Yaskawa INFORM job: OK_R2_O57-69(2)(90,0)_OK.JBI

/JOB
//NAME OK_R2_O57-69(2)(90,0)_OK
///FOLDERNAME X4
//POS
///NPOS 521,521,521,19,0,0
///TOOL 0
///POSTYPE PULSE
///PULSE
C00000=-135424,72899,29147,-3537,85342,3792
C00001=-134013,95021,61136,-4029,77105,4505
C00002=-134047,101087,71818,-4077,73656,4607
C00003=-134047,101216,72822,-4088,73105,4626
C00004=-134047,101094,71866,-4078,73630,4609
C00005=-133936,105187,77198,-4137,72460,4688
C00006=-134047,101094,71866,-4078,73630,4609
C00007=-133891,92563,58880,-4064,77236,4542
C00008=-133627,85963,47659,-4101,80754,4516
C00009=-133192,78294,50454,-10127,76922,11696
C00010=-133849,85255,61933,-10093,73405,11757
C00011=-135353,87618,67605,-9788,70974,11422
C00012=-135353,87997,69106,-9827,70255,11481
C00013=-135353,87618,67605,-9788,70974,11422
C00014=-135153,93739,75342,-9940,69404,11624
C00015=-135353,87618,67605,-9788,70974,11422
C00016=-133639,83161,60388,-10158,73308,11840
C00017=-132974,76301,49087,-10194,76769,11784
C00018=-129415,62996,33414,-11066,79991,12732
C00019=-98130,32671,61537,-45409,44339,32891
C00020=-100023,41688,73231,-46965,41628,33506
C00021=-100756,49088,84228,-49401,39255,34803
C00022=-100756,52120,89278,-50881,38240,35655
C00023=-100756,49088,84228,-49401,39255,34803
C00024=-101219,51120,86580,-49709,38764,34882
C00025=-100756,49088,84228,-49401,39255,34803
C00026=-97195,31965,62320,-46227,44186,33575
C00027=-75566,-2034,22500,-42402,86688,50389
C00028=-92276,-18388,7402,-33699,73725,46550
C00029=-92276,-17400,9548,-33822,73042,46763
C00030=-92276,-17933,8393,-33755,73407,46648
C00031=-120131,-32698,-12117,4829,66200,34356
C00032=-120131,-32114,-10702,4851,65630,34332
C00033=-120989,-32117,-10704,5006,65680,34020
C00034=-120131,-32114,-10702,4851,65630,34332
C00035=-120131,-38085,-26806,4645,72450,34604
C00036=-99101,-76935,-92016,-31014,74911,20401
C00037=-52587,-144740,-101483,-60524,64363,-65274
C00038=-46989,-65360,-59229,-62781,73103,-77672
C00039=-56832,-65466,-56421,-59287,64983,-77772
C00040=-57148,-65688,-55453,-59188,64110,-77279
C00041=-55649,-62097,-53047,-61106,66880,-78547
C00042=-57237,-59710,-51792,-60669,66110,-79037
C00043=-56277,-61326,-53166,-60831,66721,-78866
C00044=-55441,-62561,-53810,-61057,67127,-78609
C00045=-56207,-63985,-54541,-61032,66503,-78630
C00046=-55438,-62578,-53813,-61060,67126,-78606
C00047=-51973,-62323,-54701,-62406,69323,-78001
C00048=-48054,-62529,-57040,-62601,72472,-77896
C00049=-29811,-70761,-60283,-66780,94863,-53671
C00050=-30965,-22538,-31531,-67696,97011,-56857
C00051=-55044,-42598,-44870,-68563,88788,-43678
C00052=-56249,-45120,-46406,-68472,87844,-43687
C00053=-57925,-45354,-44812,-68371,86292,-43442
C00054=-57925,-45174,-43802,-68390,86084,-43215
C00055=-57925,-45354,-44812,-68371,86292,-43442
C00056=-59167,-45210,-44726,-68282,85469,-43617
C00057=-57925,-45354,-44812,-68371,86292,-43442
C00058=-55819,-44223,-45863,-68504,88181,-43684
C00059=-44722,-31045,-43816,-69927,97696,-44632
C00060=-43071,-26445,-40665,-70170,98951,-44614
C00061=-127706,-49493,-81773,19458,97242,-49666
C00062=-127020,6423,-39070,7004,99714,-51816
C00063=-127020,5137,-37554,6966,98131,-51906
C00064=-128416,4382,-35850,7239,96821,-52416
C00065=-128416,3847,-35017,7224,96041,-52460
C00066=-128416,4148,-35496,7233,96488,-52435
C00067=-130041,4566,-35136,7580,96617,-52937
C00068=-129924,4205,-34639,7545,96120,-52933
C00069=-129457,4078,-34747,7447,96082,-52788
C00070=-130190,4712,-35256,7614,96778,-52976
C00071=-128966,36168,-17458,7491,101844,-52285
C00072=-149392,-6912,-25974,9982,75562,-31317
C00073=-149173,-488,-12666,10148,70714,-31647
C00074=-149173,-326,-10897,10208,69722,-31733
C00075=-149173,-394,-11578,10184,70101,-31701
C00076=-148123,2416,-9216,9823,69962,-31333
C00077=-149173,-394,-11578,10184,70101,-31701
C00078=-152478,4885,-6741,15795,72623,-37698
C00079=-151455,3828,-7649,15488,72442,-37350
C00080=-152478,4560,-12614,15554,75946,-37261
C00081=-146445,-24647,-43161,13522,78564,-34847
C00082=-131494,-80468,-98534,7816,92108,-53678
C00083=-52065,-14099,-27709,-42253,108676,27596
C00084=-76671,-130461,-121705,-35735,90710,50834
C00085=-94829,-93442,-100428,-28991,96183,47377
C00086=-110716,-92055,-82664,-19311,98038,51285
C00087=-114275,-93352,-80055,-19461,95045,50478
C00088=-118122,-92212,-76367,-19656,92534,49497
C00089=-118129,-91398,-74848,-19645,92046,49575
C00090=-118122,-92212,-76367,-19656,92534,49497
C00091=-119808,-92271,-76389,-19753,92113,48959
C00092=-118122,-92212,-76367,-19656,92534,49497
C00093=-114499,-91094,-78376,-19482,95112,50387
C00094=-110992,-89821,-80983,-19339,98080,51178
C00095=-124454,-89651,-86550,11137,94998,-69701
C00096=-122569,-92184,-83910,11067,91866,-69331
C00097=-120652,-93960,-80852,11027,88857,-68936
C00098=-120652,-93520,-79457,11027,88237,-68992
C00099=-120652,-93960,-80852,11027,88857,-68936
C00100=-120650,-97396,-81866,11026,87737,-69033
C00101=-120652,-93960,-80852,11027,88857,-68936
C00102=-118161,-93768,-80427,10994,88357,-68121
C00103=-120652,-93960,-80852,11027,88857,-68936
C00104=-120037,-91891,-82714,11032,90945,-68539
C00105=-121981,-89592,-85452,11099,94026,-68936
C00106=-122005,-89480,-97857,11363,101580,-68254
C00107=-122005,-89427,-98101,11372,101754,-68238
C00108=-119094,-95812,-115555,-4544,90851,-20867
C00109=-116502,-111480,-109655,-18779,62868,21987
C00110=-119472,-101923,-104261,-17094,63743,20698
C00111=-121534,-96097,-100090,-16016,63743,19914
C00112=-121534,-96194,-98882,-16123,62979,20025
C00113=-112336,-84014,-94514,-26506,72534,27449
C00114=-114298,-84401,-94682,-25743,71847,26864
C00115=-121534,-96097,-100090,-16016,63743,19914
C00116=-121514,-92242,-98700,-15883,64832,19765
C00117=-121534,-96097,-100090,-16016,63743,19914
C00118=-119823,-101836,-103002,-17025,62972,20682
C00119=-116876,-111303,-108368,-18711,62117,21969
C00120=-126032,-109701,-108999,21760,66785,-27050
C00121=-122513,-101468,-103921,20079,66940,-25677
C00122=-121483,-94377,-99419,19507,67520,-25186
C00123=-121483,-94509,-98158,19621,66724,-25324
C00124=-121483,-94377,-99419,19507,67520,-25186
C00125=-119206,-94355,-99408,18489,67008,-24418
C00126=-121483,-94377,-99419,19507,67520,-25186
C00127=-121468,-91005,-98354,19362,68535,-25006
C00128=-121483,-94377,-99419,19507,67520,-25186
C00129=-124810,-108862,-107603,21303,66070,-26716
C00130=-126981,-112864,-109311,24940,61360,-29729
C00131=-123200,-104180,-104415,22777,61614,-28126
C00132=-121230,-90686,-98732,21152,64298,-26805
C00133=-121230,-90968,-97120,21351,63235,-27013
C00134=-121230,-90806,-98119,21226,63888,-26884
C00135=-118688,-90754,-98099,19926,63280,-26013
C00136=-121230,-90721,-98563,21173,64184,-26826
C00137=-121211,-84894,-96124,20922,65577,-26553
C00138=-121230,-90686,-98732,21152,64298,-26805
C00139=-121413,-93580,-100796,21282,64141,-26906
C00140=-124847,-101623,-105736,23178,64029,-28268
C00141=-120616,-95755,-103879,23668,64726,-45447
C00142=-120621,-89459,-99052,23623,64971,-45396
C00143=-102398,-78806,-99215,-137,71874,-40792
C00144=-120614,-97387,-102466,23992,63157,-45792
C00145=-122354,-96256,-100860,24938,63287,-46459
C00146=-99477,-102621,-105563,-1650,63574,-39713
C00147=-93449,-138180,-112622,-5538,49931,-36849
C00148=-85999,-163182,-115201,-11989,39587,-32297
C00149=-96470,-180165,-126119,-4784,36529,-37522
C00150=-120616,-95173,-105764,23303,89544,-42444
C00151=-107191,-96001,-89285,21702,28532,-58770
C00152=-107187,-93630,-79997,25295,24388,-60561
C00153=-107188,-92928,-77886,26213,23539,-61010
C00154=-112362,-77289,-77026,28293,40281,-63318
C00155=-107081,-94020,-78768,26067,23489,-60939
C00156=-108911,-93070,-77209,29349,23678,-62538
C00157=-100555,-91608,-91171,7273,48196,-53989
C00158=-102645,-104114,-96524,14611,51707,-64227
C00159=-108915,-55552,-83371,19664,91458,-62056
C00160=-110657,-50226,-86705,20295,96355,-61815
C00161=-107202,-93991,-108886,21178,109925,-43661
C00162=-120660,-73953,-111348,177,99224,835
C00163=-120616,-96234,-101081,-23944,56754,46777
C00164=-120615,-96493,-97034,-24670,54353,47364
C00165=-120614,-96447,-94923,-25055,53191,47662
C00166=-125343,-63714,-87611,-17170,75461,41479
C00167=-118876,-96360,-94049,-26267,53277,48431
C00168=-120612,-97621,-95709,-25094,53083,47691
C00169=-124024,-105215,-109245,-22308,82546,38090
C00170=-123496,-104488,-108175,-22872,85665,42107
C00171=-120617,-94319,-107453,-23464,90858,42123
C00172=-120617,-92878,-109780,-23521,92858,41729
C00173=-120619,-86141,-115603,-23930,99335,40429
C00174=-120619,-89012,-115558,8782,73464,77384
C00175=-120618,-92353,-112869,8941,70132,77138
C00176=-120618,-93422,-111698,9011,68877,77043
C00177=-120616,-94109,-113157,8979,69414,77085
C00178=-120318,-89311,-110489,8778,70198,77244
C00179=-120618,-93688,-111329,9132,68044,76969
C00180=-120618,-93957,-110924,9216,67187,76884
C00181=-120618,-94299,-110440,9161,65769,76809
C00182=-120618,-94831,-109599,8469,63241,76696
C00183=-120617,-95145,-109027,7071,61401,76664
C00184=-120617,-95217,-108863,5672,60665,76701
C00185=-120618,-93036,-111930,4923,63538,76718
C00186=-120618,-92960,-112001,4009,63579,76743
C00187=-120618,-92691,-112274,2433,64167,76800
C00188=-120618,-92166,-112798,840,65602,76863
C00189=-120618,-91419,-113490,-342,67708,76910
C00190=-120619,-90739,-114068,-878,69589,76936
C00191=-120619,-89701,-115007,-939,71612,76812
C00192=-120619,-88814,-115609,-873,73870,76855
C00193=-120619,-87740,-116270,-151,76574,76959
C00194=-120619,-86987,-116700,1182,78540,77121
C00195=-120619,-86782,-116823,2462,79296,77267
C00196=-120619,-90672,-114378,3278,75949,77117
C00197=-120619,-90769,-114313,4130,75889,77177
C00198=-120619,-91109,-114056,5597,75252,77256
C00199=-120618,-91719,-113544,7101,73764,77286
C00200=-120618,-92472,-112836,8259,71637,77242
C00201=-120618,-92872,-112418,8666,70405,77193
C00202=-120618,-93168,-112034,8862,69621,77111
C00203=-120618,-93422,-111698,9011,68877,77043
C00204=-120618,-92353,-112869,8941,70132,77138
C00205=-120619,-89012,-115558,8782,73464,77384
C00206=-120595,-119438,-127420,-8829,91162,8830
C00207=-129025,-103888,-99333,21372,86937,-54976
C00208=-120613,-94952,-86848,20336,81911,-52813
C00209=-120613,-94069,-83278,20415,80272,-53091
C00210=-106596,-117430,-87528,9818,57368,-33279
C00211=-120519,-95091,-83551,20421,79912,-53118
C00212=-122104,-92396,-81537,20633,80446,-53604
C00213=-112247,-111615,-87090,12951,66121,-41348
C00214=-120242,-93380,-81431,16167,85346,-56835
C00215=-120729,-92389,-78218,16226,84033,-57178
C00216=-121550,-94001,-78799,15119,86025,-61641
C00217=-122325,-96218,-79481,13215,89152,-68718
C00218=-120612,-93818,-82398,13271,91824,-67835
C00219=-120613,-94827,-86367,13308,93699,-67633
C00220=-120614,-96085,-95173,13466,98348,-67128
C00221=-120625,-105302,-100360,13404,96846,-67297
C00222=-102872,-120945,-93289,-41313,52454,35552
C00223=-111052,-89986,-73102,-36259,51528,31574
C00224=-114360,-89865,-71590,-35102,49434,30694
C00225=-117529,-82976,-67958,-32873,49251,29097
C00226=-113966,-89555,-70876,-35431,49366,30932
C00227=-115650,-91167,-72721,-34446,48930,30213
C00228=-116153,-87173,-73787,-30474,57370,33009
C00229=-115134,-90585,-78921,-28213,65812,37618
C00230=-114816,-93273,-83340,-25850,75230,43378
C00231=-115191,-85090,-71836,-25015,76673,46996
C00232=-114907,-96450,-75026,-24463,77444,52852
C00233=-115702,-94689,-74701,-23512,87260,62633
C00234=-112822,-91718,-77371,-23458,91001,62960
C00235=-109330,-92095,-80656,-23399,93677,63722
C00236=-110759,-94815,-97268,-24043,101385,61640
C00237=-25230,-87703,-86789,-41333,106155,-71905
C00238=-55862,19660,17206,-68346,89547,-53836
C00239=-59225,37567,25812,-69215,105770,-42705
C00240=-67658,42850,42597,-68102,97125,-40508
C00241=-69543,42635,44538,-68129,95346,-40204
C00242=-67599,42910,43858,-67984,96867,-40179
C00243=-68366,42138,41747,-68199,96713,-40671
C00244=-69537,42554,44453,-68130,95355,-40208
C00245=-69167,26414,28126,-68889,91591,-41841
C00246=-69430,8343,11443,-69273,87154,-43187
C00247=-70467,-11089,-4532,-69437,78929,-44678
C00248=-70464,-3151,1747,-68553,83829,-57137
C00249=-68177,-4212,-1280,-68454,85880,-57398
C00250=-65815,-3605,-3490,-68417,88124,-57797
C00251=-46513,-27715,-22241,-69125,80479,-38621
C00252=-7625,-19791,-74194,-84461,116832,-51132
C00253=-98528,-26744,-48644,-33463,55012,-18344
C00254=-108995,3085,5205,-12404,51911,-2889
C00255=-113253,15209,27106,-3834,50657,3406
C00256=-113409,21623,32322,-3755,50736,3338
C00257=-112510,30954,47444,-4478,46281,3921
C00258=-113472,24070,39362,-3899,47665,3430
C00259=-113579,25546,39455,-3805,48359,3355
C00260=-112547,30896,47385,-4459,46286,3903
C00261=-113092,30984,47541,-6567,46499,5785
C00262=-107982,35826,53096,-19952,49307,15286
C00263=-107346,38752,56151,-24065,51859,19797
C00264=-102444,58818,79888,-34511,57818,35075
C00265=-101044,76619,103296,-39601,59307,41475
C00266=-99948,73081,91706,-37976,69105,42304
C00267=-99205,63215,84174,-37575,62603,39615
C00268=-97180,56339,73463,-36771,65900,39269
C00269=-108272,10166,23438,-3323,45242,19316
C00270=-109103,10218,12469,-2549,51979,18742
C00271=-99879,30934,32617,-21980,59339,34187
C00272=-99785,30090,30578,-21838,60128,34061
C00273=-99052,29053,30612,-22206,59809,34434
C00274=-101543,26260,28122,-21325,59243,33514
C00275=-98482,32149,35009,-29284,63220,41247
C00276=-92009,66840,89116,-42947,61850,57046
C00277=-89877,62120,80876,-42077,64804,56709
C00278=-70258,15873,38394,-48666,102593,69187
C00279=-68816,9929,45318,-53577,93501,68972
C00280=-74323,28982,63484,-55349,89726,68465
C00281=-74758,1474,21309,-45746,90270,65676
C00282=-98607,12568,39814,52966,86937,78252
C00283=-98596,22842,59344,53301,82774,75788
C00284=-96296,21421,60413,54092,80731,75703
C00285=-95348,20952,60953,54433,79893,75663
C00286=-96117,19164,58324,54129,80713,75783
C00287=-95662,23434,63388,54370,79922,75521
C00288=-95503,21312,61702,54422,79811,75531
C00289=-92574,18445,54645,48983,79889,68258
C00290=-91800,17848,53101,47601,79897,67557
C00291=-92530,17999,51917,47342,80806,67673
C00292=-94302,18640,49262,46764,83033,67943
C00293=-79003,18324,29303,31626,94586,4503
C00294=-64136,40618,57122,29721,84915,83830
C00295=-62802,39067,58740,29997,82892,83805
C00296=-62255,38544,59506,30121,82059,83791
C00297=-62254,37103,56589,30066,82978,84033
C00298=-62821,40643,61741,30049,81995,83562
C00299=-59984,48909,70165,26795,84201,83115
C00300=-59410,69261,96131,25367,86084,74959
C00301=-59404,69357,96256,25356,86081,74939
C00302=-59713,70793,96681,25260,86600,74945
C00303=-60461,74839,98386,25037,87745,74932
C00304=-60470,59585,70460,25309,96249,76737
C00305=-66845,10330,41939,25249,64720,33768
C00306=-66816,16396,52426,25952,61688,33052
C00307=-66804,19142,57057,26292,60387,32730
C00308=-66058,20615,58344,26298,60142,32956
C00309=-66868,17219,53699,26035,61378,32955
C00310=-66973,19658,57552,26302,60399,32669
C00311=-66985,16895,52895,25961,61707,32992
C00312=-67015,10800,42362,25255,64752,33711
C00313=-98181,31350,57269,53093,86032,77938
C00314=-96082,29267,57446,53647,84171,77916
C00315=-95219,28523,57622,53885,83405,77901
C00316=-95917,26905,55160,53675,84199,78019
C00317=-95506,31088,60230,53837,83386,77740
C00318=-95359,28788,58259,53869,83329,77779
C00319=-92697,26913,52373,48450,83827,70215
C00320=-91994,26523,51069,47073,83939,69440
C00321=-92656,26997,50292,46905,84772,69532
C00322=-94270,28412,48618,46533,86809,69749
C00323=-79891,40483,43632,25605,98381,-17488
C00324=-64421,55368,61348,15926,95442,-62339
C00325=-63205,52871,61672,16144,93779,-62133
C00326=-62708,51961,61917,16235,93087,-62052
C00327=-62707,50761,59239,16263,94078,-61920
C00328=-63223,54241,64482,16113,92796,-62269
C00329=-60236,62044,73663,12795,94061,-63101
C00330=-59090,69141,83012,10500,94867,-70833
C00331=-59083,69182,83067,10487,94869,-70851
C00332=-59379,71028,84054,10408,95242,-70919
C00333=-60098,76023,87068,10213,96031,-71094
C00334=-60107,66003,66038,10511,103704,-70448
C00335=-66860,35146,61423,22993,49349,53528
C00336=-66834,42827,74568,24499,45535,52525
C00337=-66824,46660,80883,25305,43786,52015
C00338=-66175,48781,83167,25255,43321,52183
C00339=-66880,43946,76304,24713,45097,52378
C00340=-66970,47398,81721,25407,43702,51920
C00341=-66981,43500,75311,24586,45473,52438
C00342=-67007,35727,62031,23060,49318,53454
C00343=-87565,40229,55167,37616,76398,68031
C00344=-104252,61764,84947,51561,88394,76219
C00345=-102517,58043,82852,52038,87086,76344
C00346=-101804,56689,82195,52237,86527,76380
C00347=-102435,54601,78919,52052,87454,76595
C00348=-101993,60636,86873,52209,86091,76036
C00349=-101932,57147,83104,52210,86393,76238
C00350=-99529,53434,74771,46937,87155,68655
C00351=-98895,52660,72970,45595,87312,67859
C00352=-99433,53501,72680,45467,88010,67934
C00353=-100745,55861,72292,45181,89689,68100
C00354=-89942,52639,54543,22757,100290,-22350
C00355=-84530,60242,66965,10989,97828,-69052
C00356=-83700,56528,65849,11170,96516,-68885
C00357=-83359,55133,65530,11245,95959,-68819
C00358=-83358,53843,62725,11276,97003,-68723
C00359=-83705,58033,68848,11139,95464,-68982
C00360=-80399,62193,73871,7256,96460,-69699
C00361=-78998,67441,80988,4366,97017,-77318
C00362=-78990,67470,81028,4351,97018,-77335
C00363=-79114,69587,82331,4315,97310,-77366
C00364=-79414,75293,86196,4226,97877,-77446
C00365=-79422,65472,65446,4368,105580,-77179
C00366=-80352,27457,54566,26195,53383,48637
C00367=-80356,27473,54581,26196,53382,48635
C00368=-80357,27479,54587,26196,53382,48634
C00369=-79589,28666,55655,26054,53112,48894
C00370=-80424,25883,51570,25884,54338,48863
C00371=-80357,27479,54587,26196,53382,48634
C00372=-80356,27473,54581,26196,53382,48635
C00373=-80352,27458,54566,26195,53383,48637
C00374=-110061,-17560,-36552,26636,92274,45980
C00375=-111839,-83491,-103870,27371,99587,47031
C00376=-38426,-40229,-52385,-46753,77455,-20722
C00377=-20805,-37224,-43776,-64442,70782,-24410
C00378=-53615,-60479,-29767,-71413,48188,-35364
C00379=-53622,-60473,-29764,-71411,48184,-35366
C00380=-53625,-60471,-29763,-71411,48182,-35366
C00381=-52450,-61746,-30400,-71683,48877,-35041
C00382=-53622,-61330,-31549,-70858,48414,-35743
C00383=-53667,-60425,-29740,-73440,59962,-39458
C00384=-53705,-60384,-29719,-74506,70698,-55233
C00385=-53706,-60382,-29718,-74560,71274,-55582
C00386=-53707,-60381,-29717,-74560,71274,-55582
C00387=-53710,-60377,-29715,-74560,71273,-55583
C00388=-53701,-60384,-29719,-74560,71278,-55581
C00389=-66706,-54450,-33709,-25643,46200,-1067
C00390=-66709,-54445,-33707,-25641,46199,-1069
C00391=-65806,-56035,-34565,-26242,46218,-617
C00392=-67582,-55929,-35261,-25089,46110,-1484
C00393=-66709,-54446,-33707,-25645,46199,-1067
C00394=-66709,-54446,-33707,-25645,46199,-1067
C00395=-66709,-54447,-33708,-25641,46199,-1069
C00396=-66706,-54452,-33711,-25643,46199,-1067
C00397=-56114,-41526,-33189,-36880,64877,1074
C00398=-62492,-26274,-11536,-67617,51989,-49416
C00399=-67015,-30786,-7269,-70211,42036,-48662
C00400=-67021,-30777,-7263,-70209,42033,-48664
C00401=-67024,-30773,-7260,-70208,42031,-48665
C00402=-67025,-30771,-7259,-70208,42030,-48665
C00403=-66245,-32305,-8266,-70488,42489,-48421
C00404=-67024,-31573,-9128,-69442,42305,-49131
C00405=-67037,-30747,-7244,-72021,47713,-46269
C00406=-67060,-30703,-7215,-71923,58333,-61620
C00407=-67063,-30697,-7211,-72128,59825,-62445
C00408=-67063,-30696,-7209,-72128,59824,-62445
C00409=-67065,-30691,-7207,-72128,59824,-62445
C00410=-67053,-30709,-7218,-72128,59831,-62443
C00411=-67069,40537,9457,-57195,76262,-35492
C00412=-67067,40166,11985,-57536,75289,-34802
C00413=-67066,40064,13042,-57682,74899,-34523
C00414=-66577,38326,11242,-57768,75308,-34517
C00415=-67065,40169,11907,-57527,75318,-34822
C00416=-67072,40075,13170,-59772,79795,-32172
C00417=-67078,40614,25191,-75815,82535,-42307
C00418=-67079,40861,26780,-77445,83659,-42995
C00419=-67080,40685,25622,-77394,83811,-43275
C00420=-67085,40340,22831,-77277,84191,-43970
C00421=-67090,40073,14255,-76963,85485,-46282
C00422=-90837,-14160,-23602,-46112,79870,29092
C00423=-94881,-86110,-91503,-45134,79065,22948
C00424=-94881,-86110,-91503,-45134,79065,22948
C00425=-94881,-86110,-91503,-45134,79065,22948
C00426=-64023,-117945,-92652,-70836,68337,-59810
C00427=-77839,-63283,-64145,-64455,63318,-66711
C00428=-80052,-65654,-65354,-64094,61673,-66872
C00429=-91542,-73752,-69062,-57934,49878,-61172
C00430=-80955,-66618,-66084,-63874,61070,-67008
C00431=-80000,-68279,-65664,-64663,61180,-66324
C00432=-91387,-73280,-68839,-57922,50030,-61186
C00433=-100914,-85483,-74196,-43298,32083,-69038
C00434=-93618,-76672,-70228,-47057,37292,-67140
C00435=-87612,-64529,-64461,-48733,42323,-66403
C00436=-94575,-77342,-71004,-49651,37504,-40583
C00437=-95005,-77606,-71124,-49413,37228,-40705
C00438=-25543,-37396,-56331,-69239,85891,-31897
C00439=-172418,-62024,-69195,63943,69139,25706
C00440=-192822,-61773,-75094,68063,83874,24345
C00441=-147462,40071,30365,69170,75532,19593
C00442=-147457,40119,30415,69171,75526,19591
C00443=-147456,40127,30423,69171,75525,19590
C00444=-147721,37841,28052,69134,75813,19681
C00445=-148042,40615,30212,69143,76066,19681
C00446=-147457,40126,30423,69172,75522,19590
C00447=-147457,40126,30423,69172,75522,19590
C00448=-147457,40125,30422,69171,75526,19590
C00449=-147458,40117,30413,69171,75527,19591
C00450=-147460,40097,30392,69171,75529,19592
C00451=-134071,6209,-12454,63265,71876,23505
C00452=-134070,6228,-12438,63265,71875,23505
C00453=-134070,6235,-12431,63265,71875,23505
C00454=-134229,4110,-14261,63296,71992,23494
C00455=-134787,6570,-12855,63330,72532,23573
C00456=-134070,6235,-12432,63265,71872,23505
C00457=-134070,6235,-12432,63265,71872,23505
C00458=-134071,6233,-12433,63265,71876,23505
C00459=-134071,6226,-12439,63265,71876,23505
C00460=-134072,6208,-12455,63265,71877,23505
C00461=-134072,6180,-12479,63265,71877,23505
C00462=-130462,-25122,-37090,45275,45470,33351
C00463=-132886,-107940,-72929,67003,34868,20711
C00464=-175339,-34674,-82182,59494,83195,32396
C00465=-136096,14126,-32620,12825,85534,21552
C00466=-129268,63666,34345,-8258,78331,9264
C00467=-134681,92240,52646,-816,80365,910
C00468=-132653,94106,63405,6765,75468,-3487
C00469=-132876,98805,66718,-7260,76138,8167
C00470=-132758,95444,63654,-7290,76306,8197
C00471=-134693,106943,79821,5995,71756,-2669
C00472=-133635,106832,79602,3484,71508,162
C00473=-131960,102921,75089,-426,70802,5631
C00474=-130942,105589,75064,-6359,73995,10618
C00475=-131542,109137,74044,-11980,78923,13777
C00476=-129355,125982,76686,-9729,88276,13921
C00477=-127789,121294,71761,-15545,88654,13573
C00478=-127928,122256,73029,-17074,89645,15674
C00479=-128241,121543,71989,-17007,89844,15541
C00480=-129796,115422,63669,-14368,89697,11833
C00481=-130249,115476,63291,-14256,89876,11663
C00482=-129188,109453,52652,-14573,93397,11596
C00483=-127389,117603,65505,-15655,90606,13460
C00484=-137764,37902,26809,9618,64282,22430
C00485=-175415,-47626,-48014,65040,69542,20935
C00486=-132886,-107940,-72929,67003,34868,20711
C00487=-105972,-100304,-88890,7532,75015,-38248
C00488=-160165,-106496,-82005,21656,82129,-62098
C00489=-140609,-94579,-78221,8463,77656,-55534
C00490=-138726,-94535,-76086,8242,76183,-54976
C00491=-163390,-101496,-77356,21709,82707,-63168
C00492=-161792,-103413,-79036,21690,82331,-62654
C00493=-135933,-74368,-67331,7717,80836,-53706
C00494=-133468,-45426,-54020,7292,87230,-52484
C00495=-132807,-44691,-51453,7196,85977,-52334
C00496=-131271,-21709,-36375,6964,88353,-51682
C00497=-131369,-20934,-44335,7010,93621,-51422
C00498=-155973,16228,-7521,23092,85783,-46465
C00499=-155545,22569,6657,24866,83301,-50186
C00500=-156114,24235,11083,24511,80804,-49715
C00501=-157855,17121,1644,24703,83284,-49844
C00502=-148516,-1727,-14860,9883,71341,-31357
C00503=-147742,1394,-9472,9715,69559,-31227
C00504=-138592,3455,-7934,-8851,69391,-13105
C00505=-137116,-4730,-20716,-9180,73171,-12868
C00506=-138249,-12129,-32669,-1567,78549,-18356
C00507=-145553,-60948,-35045,47196,66698,-53129
C00508=-117087,2274,-4333,-74835,51753,34811
C00509=-120822,45639,36263,-74296,46580,35142
C00510=-132292,76688,41038,-57812,44611,25328
C00511=-133587,85399,43635,-54635,45518,23471
C00512=-134089,87151,52872,-58446,42500,25922
C00513=-133465,87868,53767,-58981,42776,26187
C00514=-134426,84651,49764,-57666,42643,25479
C00515=-134089,87030,55209,-59870,41700,26787
C00516=-134090,96417,89471,-79265,35490,37858
C00517=-134090,100042,96821,-83028,34997,39924
C00518=-133589,94413,89775,-81024,35602,38850
C00519=-132294,83338,76456,-77824,37058,37121
C00520=3643,-76224,-106676,19950,71810,76872
BC00000=138406,837384,245994
BC00001=138406,837384,245994
BC00002=138406,837384,245994
BC00003=138406,837384,245994
BC00004=138406,837384,245994
BC00005=138406,837384,245994
BC00006=138406,837384,245994
BC00007=138406,837384,245994
BC00008=138406,837384,245994
BC00009=128112,840549,330774
BC00010=128112,840549,330774
BC00011=128112,840549,330774
BC00012=128112,840549,330774
BC00013=128112,840549,330774
BC00014=128112,840549,330774
BC00015=128112,840549,330774
BC00016=128112,840549,330774
BC00017=128112,840549,330774
BC00018=128112,840549,330774
BC00019=111975,837625,420975
BC00020=111975,837625,420975
BC00021=111975,837625,420975
BC00022=111975,837625,420975
BC00023=111975,837625,420975
BC00024=111976,837626,420972
BC00025=111975,837625,420975
BC00026=111975,837625,420975
BC00027=111975,837625,420975
BC00028=111975,837625,420975
BC00029=111975,837625,420975
BC00030=111975,837625,420975
BC00031=111975,837625,420975
BC00032=111975,837625,420975
BC00033=111975,837625,420975
BC00034=111975,837625,420975
BC00035=111975,837625,420975
BC00036=111578,670431,418295
BC00037=342650,733121,86647
BC00038=339628,728489,87096
BC00039=339628,728489,87096
BC00040=339628,728489,87096
BC00041=339628,728489,87096
BC00042=339628,728489,87096
BC00043=339628,728489,87096
BC00044=339628,728489,87096
BC00045=339628,728489,87096
BC00046=339628,728489,87096
BC00047=339628,728489,87096
BC00048=339628,728489,87096
BC00049=369440,735504,90134
BC00050=369440,735504,90134
BC00051=398174,741162,97424
BC00052=398174,745386,78467
BC00053=398174,747075,70884
BC00054=398174,747075,70884
BC00055=398174,747075,70884
BC00056=398174,747075,70884
BC00057=398174,747075,70884
BC00058=398174,744503,70979
BC00059=398174,740279,89936
BC00060=398174,693649,89936
BC00061=309739,685336,89936
BC00062=309739,717578,89936
BC00063=309739,717578,89936
BC00064=309739,717578,89936
BC00065=309739,717578,89936
BC00066=309739,717578,89936
BC00067=309739,717578,89936
BC00068=309739,717578,89936
BC00069=309739,717578,89936
BC00070=309739,717578,89936
BC00071=309739,717578,89936
BC00072=311206,810481,212793
BC00073=311206,810481,212793
BC00074=311206,810481,212793
BC00075=311206,810481,212793
BC00076=311206,810481,212793
BC00077=311206,810481,212793
BC00078=311206,810481,212793
BC00079=311206,810481,212793
BC00080=311206,810481,212793
BC00081=311206,810481,212793
BC00082=309739,717578,89936
BC00083=302229,671844,714988
BC00084=365201,715179,1005006
BC00085=376221,744487,992760
BC00086=398174,770458,1075175
BC00087=398174,770458,1075175
BC00088=398174,770458,1075175
BC00089=398174,770458,1075175
BC00090=398174,770458,1075175
BC00091=398174,770458,1075175
BC00092=398174,770458,1075175
BC00093=398174,770458,1075175
BC00094=398174,770458,1075175
BC00095=395964,766843,1075175
BC00096=395964,766843,1075175
BC00097=395964,766843,1075175
BC00098=395964,766843,1075175
BC00099=395964,766843,1075175
BC00100=395964,766843,1075175
BC00101=395964,766843,1075175
BC00102=395964,766843,1075175
BC00103=395964,766843,1075175
BC00104=395964,766843,1075175
BC00105=395964,766843,1075175
BC00106=395964,766843,1075175
BC00107=395964,766843,1075175
BC00108=340614,815508,1075175
BC00109=291315,858852,1075175
BC00110=291315,858852,1075175
BC00111=291315,858852,1075175
BC00112=291315,858852,1075175
BC00113=291314,858852,1075172
BC00114=291315,858852,1075175
BC00115=291315,858852,1075175
BC00116=291315,858852,1075175
BC00117=291315,858852,1075175
BC00118=291315,858852,1075175
BC00119=291315,858852,1075175
BC00120=261388,857545,1075175
BC00121=261388,857545,1075175
BC00122=261388,857545,1075175
BC00123=261388,857545,1075175
BC00124=261388,857545,1075175
BC00125=261388,857545,1075175
BC00126=261388,857545,1075175
BC00127=261388,857545,1075175
BC00128=261388,857545,1075175
BC00129=261388,857545,1075175
BC00130=307762,841902,1075175
BC00131=307762,841902,1075175
BC00132=307762,841902,1075175
BC00133=307762,841902,1075175
BC00134=307762,841902,1075175
BC00135=307762,841902,1075175
BC00136=307762,841902,1075175
BC00137=307762,841902,1075175
BC00138=307762,841902,1075175
BC00139=307762,841902,1075175
BC00140=307762,841902,1075175
BC00141=295805,844282,1075175
BC00142=301244,847949,1075175
BC00143=301245,847950,1075171
BC00144=303420,849415,1075175
BC00145=303420,849415,1075175
BC00146=301245,847950,1075171
BC00147=301245,847950,1075171
BC00148=301245,847950,1075171
BC00149=301245,847950,1075171
BC00150=292414,841371,1075175
BC00151=232606,821958,1075175
BC00152=232627,821961,1075175
BC00153=237648,826895,1075175
BC00154=239656,828868,1075175
BC00155=239656,828868,1075175
BC00156=239656,828868,1075175
BC00157=236217,842775,1075175
BC00158=236217,842775,1075175
BC00159=236217,842775,1075175
BC00160=236217,842775,1075175
BC00161=235448,917179,1075175
BC00162=281175,871070,1075175
BC00163=310701,846914,1075175
BC00164=310711,846915,1075175
BC00165=305421,851150,1075175
BC00166=305421,851150,1075175
BC00167=303304,852843,1075175
BC00168=303304,852843,1075175
BC00169=309181,898740,1075175
BC00170=309191,897098,1075175
BC00171=311453,893904,1075175
BC00172=317069,892657,1075175
BC00173=317048,892655,1075175
BC00174=38661,866681,1075175
BC00175=39338,869210,1075175
BC00176=39608,870221,1075175
BC00177=39608,870221,1075175
BC00178=39608,870221,1075175
BC00179=44180,868724,1075175
BC00180=49942,867043,1075175
BC00181=50951,865571,1075175
BC00182=53196,863119,1075175
BC00183=56428,861533,1075175
BC00184=59256,861216,1075175
BC00185=64296,880759,1075175
BC00186=66009,881082,1075175
BC00187=68741,882049,1075175
BC00188=71304,883797,1075175
BC00189=72987,886132,1075175
BC00190=73378,888140,1075175
BC00191=51598,893084,1075175
BC00192=50729,895319,1075175
BC00193=48626,897836,1075175
BC00194=45460,899499,1075175
BC00195=42639,899847,1075175
BC00196=37245,880361,1075175
BC00197=35524,880029,1075175
BC00198=32792,879014,1075175
BC00199=30275,877177,1075175
BC00200=28702,874753,1075175
BC00201=28653,873335,1075175
BC00202=35101,871622,1075175
BC00203=39608,870221,1075175
BC00204=39338,869210,1075175
BC00205=38661,866681,1075175
BC00206=340562,849962,1075175
BC00207=386069,767337,1075175
BC00208=386069,767337,1075175
BC00209=391133,767369,1075175
BC00210=393157,767381,1075161
BC00211=393158,767383,1075175
BC00212=393158,767383,1075175
BC00213=394705,769972,1075166
BC00214=398174,775779,1075175
BC00215=389915,761514,1075175
BC00216=392098,765315,1075171
BC00217=395638,771477,1075175
BC00218=394397,772528,1075175
BC00219=391293,775155,1075175
BC00220=391272,775152,1075175
BC00221=391272,775152,1075175
BC00222=398174,746294,1075175
BC00223=398174,746296,1075175
BC00224=398174,751973,1075175
BC00225=398174,754243,1075175
BC00226=398174,754243,1075175
BC00227=398174,754243,1075175
BC00228=398174,764099,1075175
BC00229=398174,775069,1075175
BC00230=398174,788401,1075175
BC00231=398174,744649,1075175
BC00232=398174,752334,1075175
BC00233=398174,767932,1075175
BC00234=398174,768722,1075175
BC00235=398174,770697,1075175
BC00236=398174,767021,1075175
BC00237=305826,673381,1075175
BC00238=398174,694226,160353
BC00239=398174,710712,168186
BC00240=398174,710712,168186
BC00241=398174,710712,168186
BC00242=398174,710712,168186
BC00243=398174,710712,168186
BC00244=398174,710712,168186
BC00245=398174,710712,168186
BC00246=398174,710712,168186
BC00247=398174,710712,168186
BC00248=398174,710712,168186
BC00249=398174,710712,168186
BC00250=398174,710712,168186
BC00251=398174,694226,160353
BC00252=7965,694226,160353
BC00253=88425,773491,458335
BC00254=105763,819856,396590
BC00255=112823,838737,371446
BC00256=112823,838737,347276
BC00257=112823,838737,371446
BC00258=112823,838737,371446
BC00259=112823,838737,371446
BC00260=112823,838737,371446
BC00261=112823,838737,371446
BC00262=112823,838737,371446
BC00263=112823,838737,371446
BC00264=112823,838737,371446
BC00265=112823,838737,371446
BC00266=112823,842247,331141
BC00267=112823,838737,371446
BC00268=112823,838737,371446
BC00269=95917,841923,362982
BC00270=95917,841923,278580
BC00271=95918,841923,278577
BC00272=95918,841923,278577
BC00273=95918,841923,278577
BC00274=95918,841923,278577
BC00275=95918,841923,278580
BC00276=95917,841923,362982
BC00277=95917,841923,362982
BC00278=95917,841923,362982
BC00279=95917,841923,362982
BC00280=95917,841923,362982
BC00281=95917,841923,362982
BC00282=113760,802727,443486
BC00283=113760,802727,443486
BC00284=113760,802727,443486
BC00285=113760,802727,443486
BC00286=113760,802727,443486
BC00287=113760,802727,443486
BC00288=113760,802727,443486
BC00289=113760,802727,443486
BC00290=113760,802727,443486
BC00291=113760,802727,443486
BC00292=113760,802727,443486
BC00293=105225,809384,420294
BC00294=71151,822459,422634
BC00295=71151,822459,422634
BC00296=71151,822459,422634
BC00297=71151,822459,422634
BC00298=71151,822459,422634
BC00299=71151,822459,422634
BC00300=71151,822459,422634
BC00301=71151,822459,422634
BC00302=71151,822459,422634
BC00303=71151,822459,422634
BC00304=71151,822459,422634
BC00305=83716,796230,577321
BC00306=83716,796230,577321
BC00307=83716,796230,577321
BC00308=83716,796230,577321
BC00309=83716,796230,577321
BC00310=83716,796230,577321
BC00311=83716,796230,577321
BC00312=83716,796230,577321
BC00313=107468,821574,386040
BC00314=107468,821574,386040
BC00315=107468,821574,386040
BC00316=107468,821574,386040
BC00317=107468,821574,386040
BC00318=107468,821574,386040
BC00319=107468,821574,386040
BC00320=107468,821574,386040
BC00321=107468,821574,386040
BC00322=107468,821574,386040
BC00323=98517,821001,368440
BC00324=79840,837992,369859
BC00325=79840,837992,369859
BC00326=79840,837992,369859
BC00327=79840,837992,369859
BC00328=79840,837992,369859
BC00329=79840,837992,369859
BC00330=79840,837992,369859
BC00331=79840,837992,369859
BC00332=79840,837992,369859
BC00333=79840,837992,369859
BC00334=79840,837992,369859
BC00335=56247,787784,530537
BC00336=56247,787784,530537
BC00337=56247,787784,530537
BC00338=56247,787784,530537
BC00339=56247,787784,530537
BC00340=56247,787784,530537
BC00341=56247,787784,530537
BC00342=56247,787784,530537
BC00343=90098,809263,432129
BC00344=117602,826714,352172
BC00345=117602,826714,352172
BC00346=117602,826714,352172
BC00347=117602,826714,352172
BC00348=117602,826714,352172
BC00349=117602,826714,352172
BC00350=117602,826714,352172
BC00351=117602,826714,352172
BC00352=117602,826714,352172
BC00353=117602,826714,352172
BC00354=126877,832651,364221
BC00355=131515,835619,370246
BC00356=131515,835619,370246
BC00357=131515,835619,370246
BC00358=131515,835619,370246
BC00359=131515,835619,370246
BC00360=131515,835619,370246
BC00361=131515,835619,370246
BC00362=131515,835619,370246
BC00363=131515,835619,370246
BC00364=131515,835619,370246
BC00365=131515,835619,370246
BC00366=90780,809429,536518
BC00367=91468,810120,509844
BC00368=91743,810396,499175
BC00369=91743,810396,499175
BC00370=91743,810396,499175
BC00371=91745,811011,499181
BC00372=91470,810734,509851
BC00373=90782,810043,536525
BC00374=90780,809429,536518
BC00375=90780,677587,536518
BC00376=122178,711426,262582
BC00377=129566,724478,198127
BC00378=152481,738510,229723
BC00379=153188,743935,210842
BC00380=153471,746105,203290
BC00381=153471,746105,203290
BC00382=153471,746105,203290
BC00383=178419,747743,194040
BC00384=198738,754799,174592
BC00385=199704,755257,173467
BC00386=201481,753446,179748
BC00387=205924,748918,195450
BC00388=205914,748916,222334
BC00389=140861,743664,275053
BC00390=142200,745983,269639
BC00391=142200,745983,269639
BC00392=142200,745983,269639
BC00393=141326,745985,265401
BC00394=139461,745998,256423
BC00395=138579,746008,252202
BC00396=137239,743689,257616
BC00397=140861,743664,275053
BC00398=158142,738296,276224
BC00399=157676,736172,283618
BC00400=157686,736173,256734
BC00401=156866,741594,237889
BC00402=156538,743762,230351
BC00403=156538,743762,230351
BC00404=156538,743762,230351
BC00405=167187,744647,226440
BC00406=187251,751680,220156
BC00407=189813,752792,218066
BC00408=191590,750981,224347
BC00409=196033,746452,240049
BC00410=196012,746450,293816
BC00411=131888,717539,53
BC00412=131068,722959,53
BC00413=130740,725127,53
BC00414=130740,725127,53
BC00415=130740,725127,53
BC00416=139307,729508,53
BC00417=158758,734252,53
BC00418=161265,735929,53
BC00419=163042,734117,53
BC00420=167485,729589,53
BC00421=167464,729587,53
BC00422=109122,808327,293501
BC00423=110915,803765,284066
BC00424=110915,697318,284066
BC00425=308726,697318,147266
BC00426=398174,705389,4619
BC00427=398174,702811,16248
BC00428=398174,707203,53
BC00429=398174,705653,53
BC00430=398174,708960,53
BC00431=398174,708960,53
BC00432=398174,705653,53
BC00433=398174,705653,53
BC00434=398174,705653,53
BC00435=398174,705653,53
BC00436=398174,698596,1447
BC00437=398174,692515,17689
BC00438=264874,694777,10629
BC00439=251942,672671,69662
BC00440=174905,676397,197036
BC00441=246048,666220,100031
BC00442=249809,671543,85513
BC00443=251313,673683,79706
BC00444=251313,673683,79706
BC00445=251313,673683,79706
BC00446=250438,673684,75469
BC00447=248573,673697,66491
BC00448=247692,673708,62269
BC00449=246187,671568,68076
BC00450=242426,666217,82593
BC00451=199516,725910,40957
BC00452=203277,731261,26440
BC00453=204782,733401,20633
BC00454=204782,733401,20633
BC00455=204782,733401,20633
BC00456=203934,733402,16530
BC00457=202042,733415,7418
BC00458=201188,733426,3329
BC00459=199684,731286,9136
BC00460=195923,725935,23654
BC00461=195902,725933,77421
BC00462=197406,728073,71614
BC00463=197406,671867,269361
BC00464=197406,671867,269361
BC00465=156718,775147,252165
BC00466=132577,836422,356218
BC00467=132577,836422,204582
BC00468=132577,836422,241964
BC00469=132577,836422,241964
BC00470=132577,836422,241964
BC00471=132577,836422,241964
BC00472=132577,836422,241964
BC00473=132577,836422,241964
BC00474=132577,836422,222331
BC00475=132577,836422,186039
BC00476=117803,830955,65927
BC00477=113819,828411,65917
BC00478=106531,823737,65871
BC00479=106531,823737,65871
BC00480=106531,823737,65871
BC00481=106531,823737,65871
BC00482=106531,823737,65871
BC00483=111823,818035,92310
BC00484=155346,771391,566288
BC00485=197406,671867,536806
BC00486=197406,671867,269361
BC00487=259574,750536,237143
BC00488=311205,810481,212796
BC00489=311205,810481,212796
BC00490=311205,810481,212796
BC00491=311205,810481,212796
BC00492=311205,810481,212796
BC00493=311205,810481,212796
BC00494=311205,810481,212796
BC00495=311205,810481,212796
BC00496=311205,810481,212796
BC00497=311205,810481,212796
BC00498=311206,810481,212793
BC00499=311206,810481,212793
BC00500=311206,810481,212793
BC00501=311206,810481,212793
BC00502=311206,810481,212793
BC00503=311206,810481,212793
BC00504=311206,810481,212793
BC00505=311206,810481,212793
BC00506=315649,791685,239699
BC00507=344285,670537,413125
BC00508=148456,753848,427487
BC00509=149313,803884,512961
BC00510=149313,803884,314593
BC00511=149313,803884,267132
BC00512=149313,803884,314593
BC00513=149313,803884,314593
BC00514=149313,803884,314593
BC00515=149313,803884,314593
BC00516=149313,803884,314593
BC00517=149313,803884,314593
BC00518=149313,803884,314593
BC00519=149313,803884,314593
BC00520=199464,674570,1075173
EC00000=798156,1112951
EC00001=798156,1112951
EC00002=798156,1112951
EC00003=798156,1112951
EC00004=798156,1112951
EC00005=798156,1112951
EC00006=798156,1112951
EC00007=798156,1112951
EC00008=798156,1112951
EC00009=798156,1112951
EC00010=798156,1112951
EC00011=798156,1112951
EC00012=798156,1112951
EC00013=798156,1112951
EC00014=798156,1112951
EC00015=798156,1112951
EC00016=798156,1112951
EC00017=798156,1112951
EC00018=798156,1112951
EC00019=798156,1112951
EC00020=798156,1112951
EC00021=798156,1112951
EC00022=798156,1112951
EC00023=798156,1112951
EC00024=798155,1112950
EC00025=798156,1112951
EC00026=798156,1112951
EC00027=798156,1112951
EC00028=798156,1112951
EC00029=798156,1112951
EC00030=798156,1112951
EC00031=798156,1112951
EC00032=798156,1112951
EC00033=798156,1112951
EC00034=798156,1112951
EC00035=798156,1112951
EC00036=798156,1112951
EC00037=798156,1112951
EC00038=798156,1112951
EC00039=798156,1112951
EC00040=798156,1112951
EC00041=798156,1112951
EC00042=798156,1112951
EC00043=798156,1112951
EC00044=798156,1112951
EC00045=798156,1112951
EC00046=798156,1112951
EC00047=798156,1112951
EC00048=798156,1112951
EC00049=798156,1112951
EC00050=798156,1112951
EC00051=798156,1112951
EC00052=798156,1112951
EC00053=798156,1112951
EC00054=798156,1112951
EC00055=798156,1112951
EC00056=798156,1112951
EC00057=798156,1112951
EC00058=798156,1112951
EC00059=798156,1112951
EC00060=798156,1112951
EC00061=798156,1112951
EC00062=798156,1112951
EC00063=798156,1112951
EC00064=798156,1112951
EC00065=798156,1112951
EC00066=798156,1112951
EC00067=798156,1112951
EC00068=798156,1112951
EC00069=798156,1112951
EC00070=798156,1112951
EC00071=798156,1112951
EC00072=798155,1112950
EC00073=798155,1112950
EC00074=798155,1112950
EC00075=798155,1112950
EC00076=798155,1112950
EC00077=798155,1112950
EC00078=798155,1112950
EC00079=798155,1112950
EC00080=798155,1112950
EC00081=798155,1112950
EC00082=798156,1112951
EC00083=910680,1112951
EC00084=953239,1112951
EC00085=960687,1112951
EC00086=975524,1112951
EC00087=975524,1112951
EC00088=975524,1112951
EC00089=975524,1112951
EC00090=975524,1112951
EC00091=975524,1112951
EC00092=975524,1112951
EC00093=975524,1112951
EC00094=975524,1112951
EC00095=975524,1112951
EC00096=975524,1112951
EC00097=975524,1112951
EC00098=975524,1112951
EC00099=975524,1112951
EC00100=975524,1112951
EC00101=975524,1112951
EC00102=975524,1112951
EC00103=975524,1112951
EC00104=975524,1112951
EC00105=975524,1112951
EC00106=975524,1112951
EC00107=975524,1112951
EC00108=975524,1112951
EC00109=975524,1112951
EC00110=975524,1112951
EC00111=975524,1112951
EC00112=975524,1112951
EC00113=975521,1112950
EC00114=975524,1112951
EC00115=975524,1112951
EC00116=975524,1112951
EC00117=975524,1112951
EC00118=975524,1112951
EC00119=975524,1112951
EC00120=975524,1112951
EC00121=975524,1112951
EC00122=975524,1112951
EC00123=975524,1112951
EC00124=975524,1112951
EC00125=975524,1112951
EC00126=975524,1112951
EC00127=975524,1112951
EC00128=975524,1112951
EC00129=975524,1112951
EC00130=975524,1112951
EC00131=975524,1112951
EC00132=975524,1112951
EC00133=975524,1112951
EC00134=975524,1112951
EC00135=975524,1112951
EC00136=975524,1112951
EC00137=975524,1112951
EC00138=975524,1112951
EC00139=975524,1112951
EC00140=975524,1112951
EC00141=975524,1112951
EC00142=975524,1112951
EC00143=975521,1112951
EC00144=975524,1112951
EC00145=975524,1112951
EC00146=975521,1112951
EC00147=975521,1112951
EC00148=975521,1112951
EC00149=975521,1112951
EC00150=975524,1112951
EC00151=975524,1112951
EC00152=975524,1112951
EC00153=975524,1112951
EC00154=975524,1112951
EC00155=975524,1112951
EC00156=975524,1112951
EC00157=975524,1112951
EC00158=975524,1112951
EC00159=975524,1112951
EC00160=975524,1112951
EC00161=975524,1112951
EC00162=975524,1112951
EC00163=975524,1112951
EC00164=975524,1112951
EC00165=975524,1112951
EC00166=975524,1112951
EC00167=975524,1112951
EC00168=975524,1112951
EC00169=975524,1112951
EC00170=975524,1112951
EC00171=975524,1112951
EC00172=975524,1112951
EC00173=975524,1112951
EC00174=975524,1112951
EC00175=975524,1112951
EC00176=975524,1112951
EC00177=975524,1112951
EC00178=975524,1112951
EC00179=975524,1112951
EC00180=975524,1112951
EC00181=975524,1112951
EC00182=975524,1112951
EC00183=975524,1112951
EC00184=975524,1112951
EC00185=975524,1112951
EC00186=975524,1112951
EC00187=975524,1112951
EC00188=975524,1112951
EC00189=975524,1112951
EC00190=975524,1112951
EC00191=975524,1112951
EC00192=975524,1112951
EC00193=975524,1112951
EC00194=975524,1112951
EC00195=975524,1112951
EC00196=975524,1112951
EC00197=975524,1112951
EC00198=975524,1112951
EC00199=975524,1112951
EC00200=975524,1112951
EC00201=975524,1112951
EC00202=975524,1112951
EC00203=975524,1112951
EC00204=975524,1112951
EC00205=975524,1112951
EC00206=975524,1112951
EC00207=975524,1112951
EC00208=975524,1112951
EC00209=975524,1112951
EC00210=975512,1112947
EC00211=975524,1112951
EC00212=975524,1112951
EC00213=975515,1112948
EC00214=975524,1112951
EC00215=975524,1112951
EC00216=975521,1112950
EC00217=975524,1112951
EC00218=975524,1112951
EC00219=975524,1112951
EC00220=975524,1112951
EC00221=975524,1112951
EC00222=975524,1112951
EC00223=975524,1112951
EC00224=975524,1112951
EC00225=975524,1112951
EC00226=975524,1112951
EC00227=975524,1112951
EC00228=975524,1112951
EC00229=975524,1112951
EC00230=975524,1112951
EC00231=975524,1112951
EC00232=975524,1112951
EC00233=975524,1112951
EC00234=975524,1112951
EC00235=975524,1112951
EC00236=975524,1112951
EC00237=975524,1112951
EC00238=798156,1112951
EC00239=798156,1112951
EC00240=798156,1112951
EC00241=798156,1112951
EC00242=798156,1112951
EC00243=798156,1112951
EC00244=798156,1112951
EC00245=798156,1112951
EC00246=798156,1112951
EC00247=798156,1112951
EC00248=798156,1112951
EC00249=798156,1112951
EC00250=798156,1112951
EC00251=798156,1112951
EC00252=798156,1112951
EC00253=798156,1112951
EC00254=798156,1112951
EC00255=798156,1112951
EC00256=798156,1112951
EC00257=798156,1112951
EC00258=798156,1112951
EC00259=798156,1112951
EC00260=798156,1112951
EC00261=798156,1112951
EC00262=798156,1112951
EC00263=798156,1112951
EC00264=798156,1112951
EC00265=798156,1112951
EC00266=798155,1112950
EC00267=798156,1112951
EC00268=798156,1112951
EC00269=798156,1112951
EC00270=798156,1112951
EC00271=798155,1112950
EC00272=798155,1112950
EC00273=798155,1112950
EC00274=798155,1112950
EC00275=798155,1112950
EC00276=798156,1112951
EC00277=798156,1112951
EC00278=798156,1112951
EC00279=798156,1112951
EC00280=798156,1112951
EC00281=798156,1112951
EC00282=798156,1112951
EC00283=798156,1112951
EC00284=798156,1112951
EC00285=798156,1112951
EC00286=798156,1112951
EC00287=798156,1112951
EC00288=798156,1112951
EC00289=798156,1112951
EC00290=798156,1112951
EC00291=798156,1112951
EC00292=798156,1112951
EC00293=798156,1112951
EC00294=798156,1112951
EC00295=798156,1112951
EC00296=798156,1112951
EC00297=798156,1112951
EC00298=798156,1112951
EC00299=798156,1112951
EC00300=798156,1112951
EC00301=798156,1112951
EC00302=798156,1112951
EC00303=798156,1112951
EC00304=798156,1112951
EC00305=798156,1112951
EC00306=798156,1112951
EC00307=798156,1112951
EC00308=798156,1112951
EC00309=798156,1112951
EC00310=798156,1112951
EC00311=798156,1112951
EC00312=798156,1112951
EC00313=798156,1112951
EC00314=798156,1112951
EC00315=798156,1112951
EC00316=798156,1112951
EC00317=798156,1112951
EC00318=798156,1112951
EC00319=798156,1112951
EC00320=798156,1112951
EC00321=798156,1112951
EC00322=798156,1112951
EC00323=798156,1112951
EC00324=798156,1112951
EC00325=798156,1112951
EC00326=798156,1112951
EC00327=798156,1112951
EC00328=798156,1112951
EC00329=798156,1112951
EC00330=798156,1112951
EC00331=798156,1112951
EC00332=798156,1112951
EC00333=798156,1112951
EC00334=798156,1112951
EC00335=798156,1112951
EC00336=798156,1112951
EC00337=798156,1112951
EC00338=798156,1112951
EC00339=798156,1112951
EC00340=798156,1112951
EC00341=798156,1112951
EC00342=798156,1112951
EC00343=798156,1112951
EC00344=798156,1112951
EC00345=798156,1112951
EC00346=798156,1112951
EC00347=798156,1112951
EC00348=798156,1112951
EC00349=798156,1112951
EC00350=798156,1112951
EC00351=798156,1112951
EC00352=798156,1112951
EC00353=798156,1112951
EC00354=798156,1112951
EC00355=798156,1112951
EC00356=798156,1112951
EC00357=798156,1112951
EC00358=798156,1112951
EC00359=798156,1112951
EC00360=798156,1112951
EC00361=798156,1112951
EC00362=798156,1112951
EC00363=798156,1112951
EC00364=798156,1112951
EC00365=798156,1112951
EC00366=798156,1112951
EC00367=798156,1112951
EC00368=798156,1112951
EC00369=798156,1112951
EC00370=798156,1112951
EC00371=798156,1112951
EC00372=798156,1112951
EC00373=798156,1112951
EC00374=798156,1112951
EC00375=798156,1112951
EC00376=798156,1112951
EC00377=798156,1112951
EC00378=798156,1112951
EC00379=798156,1112951
EC00380=798156,1112951
EC00381=798156,1112951
EC00382=798156,1112951
EC00383=798156,1112951
EC00384=798156,1112951
EC00385=798156,1112951
EC00386=798156,1112951
EC00387=798156,1112951
EC00388=798156,1112951
EC00389=798156,1112951
EC00390=798156,1112951
EC00391=798156,1112951
EC00392=798156,1112951
EC00393=798156,1112951
EC00394=798156,1112951
EC00395=798156,1112951
EC00396=798156,1112951
EC00397=798156,1112951
EC00398=798156,1112951
EC00399=798156,1112951
EC00400=798156,1112951
EC00401=798156,1112951
EC00402=798156,1112951
EC00403=798156,1112951
EC00404=798156,1112951
EC00405=798156,1112951
EC00406=798156,1112951
EC00407=798156,1112951
EC00408=798156,1112951
EC00409=798156,1112951
EC00410=798156,1112951
EC00411=798156,1112951
EC00412=798156,1112951
EC00413=798156,1112951
EC00414=798156,1112951
EC00415=798156,1112951
EC00416=798156,1112951
EC00417=798156,1112951
EC00418=798156,1112951
EC00419=798156,1112951
EC00420=798156,1112951
EC00421=798156,1112951
EC00422=798156,1112951
EC00423=798156,1112951
EC00424=798156,1112951
EC00425=798156,1112951
EC00426=798156,1112951
EC00427=798156,1112951
EC00428=798156,1112951
EC00429=798156,1112951
EC00430=798156,1112951
EC00431=798156,1112951
EC00432=798156,1112951
EC00433=798156,1112951
EC00434=798156,1112951
EC00435=798156,1112951
EC00436=798156,1112951
EC00437=798156,1112951
EC00438=798156,1112951
EC00439=798156,1112951
EC00440=798156,1112951
EC00441=798156,1112951
EC00442=798156,1112951
EC00443=798156,1112951
EC00444=798156,1112951
EC00445=798156,1112951
EC00446=798156,1112951
EC00447=798156,1112951
EC00448=798156,1112951
EC00449=798156,1112951
EC00450=798156,1112951
EC00451=798156,1112951
EC00452=798156,1112951
EC00453=798156,1112951
EC00454=798156,1112951
EC00455=798156,1112951
EC00456=798156,1112951
EC00457=798156,1112951
EC00458=798156,1112951
EC00459=798156,1112951
EC00460=798156,1112951
EC00461=798156,1112951
EC00462=798156,1112951
EC00463=798156,1112951
EC00464=798156,1112951
EC00465=798155,1112951
EC00466=798156,1112951
EC00467=798156,1112951
EC00468=798156,1112951
EC00469=798156,1112951
EC00470=798156,1112951
EC00471=798156,1112951
EC00472=798156,1112951
EC00473=798156,1112951
EC00474=798156,1112951
EC00475=798156,1112951
EC00476=798156,1112951
EC00477=798156,1112951
EC00478=798156,1112951
EC00479=798156,1112951
EC00480=798156,1112951
EC00481=798156,1112951
EC00482=798156,1112951
EC00483=798156,1112951
EC00484=798156,1112951
EC00485=798156,1112951
EC00486=798156,1112951
EC00487=798156,1112951
EC00488=798156,1112951
EC00489=798156,1112951
EC00490=798156,1112951
EC00491=798156,1112951
EC00492=798156,1112951
EC00493=798156,1112951
EC00494=798156,1112951
EC00495=798156,1112951
EC00496=798156,1112951
EC00497=798156,1112951
EC00498=798155,1112950
EC00499=798155,1112950
EC00500=798155,1112950
EC00501=798155,1112950
EC00502=798155,1112950
EC00503=798155,1112950
EC00504=798155,1112950
EC00505=798155,1112950
EC00506=798155,1112950
EC00507=798156,1112951
EC00508=798156,1112951
EC00509=798156,1112951
EC00510=798156,1112951
EC00511=798156,1112951
EC00512=798156,1112951
EC00513=798156,1112951
EC00514=798156,1112951
EC00515=798156,1112951
EC00516=798156,1112951
EC00517=798156,1112951
EC00518=798156,1112951
EC00519=798156,1112951
EC00520=798155,1112950
///POSTYPE BASE
///RECTAN
///RCONF 0,0,0,0,0,0,0,0,0,0,0,0,0,0,0,0,0,0,0,0,0,0,0,0
P00006=0.222,-3.123,-1.508,0.0000,0.0000,0.0000
P00021=-0.225,-6.128,-0.405,0.0000,0.0000,0.0000
P00022=0.222,-3.123,-1.508,0.0000,0.0000,0.0000
P00023=0.143,-0.036,0.682,0.0000,0.0000,0.0000
P00024=0.145,-0.552,1.326,0.0000,0.0000,0.0000
P00025=-2.003,0.006,0.728,0.0000,0.0000,0.0000
P00026=0.562,-0.002,-0.337,0.0000,0.0000,0.0000
P00027=-0.746,0.015,-9.096,0.0000,0.0000,0.0000
P00031=1.853,-0.001,-1.549,0.0000,0.0000,0.0000
P00032=1.957,0.503,-7.217,0.0000,0.0000,0.0000
P00041=0.192,3.924,0.305,0.0000,0.0000,0.0000
P00042=-0.217,1.941,0.413,0.0000,0.0000,0.0000
P00043=-0.044,-1.937,1.197,0.0000,0.0000,0.0000
P00044=0.687,-2.322,1.156,0.0000,0.0000,0.0000
P00045=-0.068,-0.810,1.603,0.0000,0.0000,0.0000
P00046=0.799,0.043,1.292,0.0000,0.0000,0.0000
P00088=-2.376,0.094,2.453,0.0000,0.0000,0.0000
P00089=5.697,-3.100,-1.263,0.0000,0.0000,0.0000
P00090=0.184,3.539,2.293,0.0000,0.0000,0.0000
//INST
///DATE 2025/02/07 12:19
///ATTR SC,RW
///GROUP1 RB1,BS1
///GROUP2 ST1
NOP
'OK_r2_O57-69(2)(90,0)2
'Down
SFTOF3D
MOVJ C00000 BC00000 VJ=100.00  +MOVJ EC00000 VJ=100.00
MOVL C00001 BC00001 V=400.0  +MOVJ EC00001 VJ=100.00
SMOVL C00002 BC00002 V=166.7  +MOVJ EC00002
SREFP 3 C00003 BC00003  +REFP EC00003
CALL JOB:SEARCH-R1-S13D
SET P026 P006
SFTON3D P026
SMOVL C00004 BC00004 V=166.7  +MOVJ EC00004
SREFP 3 C00005 BC00005  +REFP EC00005
CALL JOB:SEARCH-R1-S13D
SET P026 P006
SFTON3D P026
SMOVL C00006 BC00006 V=166.7  +MOVJ EC00006
MOVL C00007 BC00007 V=400.0  +MOVJ EC00007 VJ=100.00
MOVL C00008 BC00008 V=1000.0  +MOVJ EC00008 VJ=100.00
'Path S3529
SFTOF3D
MOVJ C00009 BC00009 VJ=100.00  +MOVJ EC00009 VJ=100.00
MOVL C00010 BC00010 V=400.0  +MOVJ EC00010 VJ=100.00
SMOVL C00011 BC00011 V=166.7  +MOVJ EC00011
SREFP 3 C00012 BC00012  +REFP EC00012
CALL JOB:SEARCH-R1-S13D
SET P027 P006
SFTON3D P027
SMOVL C00013 BC00013 V=166.7  +MOVJ EC00013
SREFP 3 C00014 BC00014  +REFP EC00014
CALL JOB:SEARCH-R1-S13D
SET P027 P006
SFTON3D P027
SMOVL C00015 BC00015 V=166.7  +MOVJ EC00015
MOVL C00016 BC00016 V=400.0  +MOVJ EC00016 VJ=100.00
MOVL C00017 BC00017 V=1000.0  +MOVJ EC00017 VJ=100.00
MOVL C00018 BC00018 V=1000.0  +MOVJ EC00018 VJ=100.00
'Path S3530
SFTOF3D
MOVJ C00019 BC00019 VJ=100.00  +MOVJ EC00019 VJ=100.00
COMM PAUSE
COMM MOVL C00020 BC00020 V=400.0  +MOVJ EC00020 VJ=100.00
COMM SMOVL C00021 BC00021 V=166.7  +MOVJ EC00021
COMM SREFP 3 C00022 BC00022  +REFP EC00022
COMM CALL JOB:SEARCH-R1-S13D
COMM SET P022 P006
COMM SFTON3D P022
COMM SMOVL C00023 BC00023 V=166.7  +MOVJ EC00023
COMM SREFP 3 C00024 BC00024  +REFP EC00024
COMM CALL JOB:SEARCH-R1-S13D
COMM SET P022 P006
COMM SFTON3D P022
COMM SMOVL C00025 BC00025 V=166.7  +MOVJ EC00025
COMM SFTOF3D
COMM MOVL C00026 BC00026 V=1000.0  +MOVJ EC00026 VJ=100.00
COMM PAUSE
SMOVL C00027 BC00027 V=1000.0  +MOVJ EC00027
SMOVL C00028 BC00028 V=166.7  +MOVJ EC00028
SREFP 3 C00029 BC00029  +REFP EC00029
CALL JOB:SEARCH-R1-S13D
SET P088 P006
SFTON3D P088
SMOVL C00030 BC00030 V=166.7  +MOVJ EC00030
SMOVL C00031 BC00031 V=166.7  +MOVJ EC00031
SMOVL C00032 BC00032 V=166.7  +MOVJ EC00032
SREFP 3 C00033 BC00033  +REFP EC00033
CALL JOB:SEARCH-R1-S13D
SET P088 P006
SFTON3D P088
SMOVL C00034 BC00034 V=166.7  +MOVJ EC00034
SFTOF3D
SMOVL C00035 BC00035 V=1000.0  +MOVJ EC00035
MOVJ C00036 BC00036 VJ=100.00  +MOVJ EC00036 VJ=100.00
MOVJ C00037 BC00037 VJ=100.00  +MOVJ EC00037 VJ=100.00
MOVL C00038 BC00038 V=400.0  +MOVJ EC00038 VJ=100.00
SMOVL C00039 BC00039 V=133.3  +MOVJ EC00039
SREFP 3 C00040 BC00040  +REFP EC00040
CALL JOB:SEARCH-R1-S13D
SET P021 P006
SFTON3D P021
SMOVL C00041 BC00041 V=166.7  +MOVJ EC00041
SREFP 3 C00042 BC00042  +REFP EC00042
CALL JOB:SEARCH-R1-S13D
SET P021 P006
SFTON3D P021
SMOVL C00043 BC00043 V=166.7  +MOVJ EC00043
SMOVL C00044 BC00044 V=166.7  +MOVJ EC00044
SREFP 3 C00045 BC00045  +REFP EC00045
CALL JOB:SEARCH-R1-S13D
SET P021 P006
SFTON3D P021
SMOVL C00046 BC00046 V=166.7  +MOVJ EC00046
MOVL C00047 BC00047 V=400.0  +MOVJ EC00047 VJ=100.00
MOVL C00048 BC00048 V=1000.0  +MOVJ EC00048 VJ=100.00
MOVJ C00049 BC00049 VJ=100.00  +MOVJ EC00049 VJ=100.00
MOVJ C00050 BC00050 VJ=100.00  +MOVJ EC00050 VJ=100.00
'Path S3538
SFTOF3D
MOVJ C00051 BC00051 VJ=100.00  +MOVJ EC00051 VJ=100.00
MOVL C00052 BC00052 V=400.0  +MOVJ EC00052 VJ=100.00
SMOVL C00053 BC00053 V=166.7  +MOVJ EC00053
SREFP 3 C00054 BC00054  +REFP EC00054
CALL JOB:SEARCH-R1-S13D
SET P032 P006
SFTON3D P032
SMOVL C00055 BC00055 V=166.7  +MOVJ EC00055
SREFP 3 C00056 BC00056  +REFP EC00056
CALL JOB:SEARCH-R1-S13D
SET P032 P006
SFTON3D P032
SMOVL C00057 BC00057 V=166.7  +MOVJ EC00057
SFTOF3D
MOVL C00058 BC00058 V=400.0  +MOVJ EC00058 VJ=100.00
MOVL C00059 BC00059 V=1000.0  +MOVJ EC00059 VJ=100.00
MOVJ C00060 BC00060 VJ=100.00  +MOVJ EC00060 VJ=100.00
MOVJ C00061 BC00061 VJ=100.00  +MOVJ EC00061 VJ=100.00
COMM PAUSE
COMM MOVJ C00062 BC00062 VJ=100.00  +MOVJ EC00062 VJ=100.00
COMM SMOVL C00063 BC00063 V=1000.0  +MOVJ EC00063
COMM SMOVL C00064 BC00064 V=166.7  +MOVJ EC00064
COMM SREFP 3 C00065 BC00065  +REFP EC00065
COMM CALL JOB:SEARCH-R1-S13D
COMM SET P089 P006
COMM SFTON3D P089
COMM SMOVL C00066 BC00066 V=166.7  +MOVJ EC00066
COMM SMOVL C00067 BC00067 V=166.7  +MOVJ EC00067
COMM SMOVL C00068 BC00068 V=166.7  +MOVJ EC00068
COMM SREFP 3 C00069 BC00069  +REFP EC00069
COMM CALL JOB:SEARCH-R1-S13D
COMM SET P089 P006
COMM SFTON3D P089
COMM SMOVL C00070 BC00070 V=166.7  +MOVJ EC00070
COMM SFTOF3D
SMOVL C00071 BC00071 V=1000.0  +MOVJ EC00071
SMOVL C00072 BC00072 V=1000.0  +MOVJ EC00072
SMOVL C00073 BC00073 V=166.7  +MOVJ EC00073
SREFP 3 C00074 BC00074  +REFP EC00074
CALL JOB:SEARCH-R1-S13D
SET P090 P006
SFTON3D P090
SMOVL C00075 BC00075 V=166.7  +MOVJ EC00075
SREFP 3 C00076 BC00076  +REFP EC00076
CALL JOB:SEARCH-R1-S13D
SET P090 P006
SFTON3D P090
SMOVL C00077 BC00077 V=166.7  +MOVJ EC00077
SMOVL C00078 BC00078 V=166.7  +MOVJ EC00078
SREFP 3 C00079 BC00079  +REFP EC00079
CALL JOB:SEARCH-R1-S13D
SET P090 P006
SFTON3D P090
SMOVL C00080 BC00080 V=250.0  +MOVJ EC00080
SFTOF3D
SMOVL C00081 BC00081 V=1000.0  +MOVJ EC00081
SMOVL C00082 BC00082 V=1000.0  +MOVJ EC00082
MOVJ C00083 BC00083 VJ=100.00  +MOVJ EC00083 VJ=100.00
'Up
MOVJ C00084 BC00084 VJ=100.00  +MOVJ EC00084 VJ=100.00
MOVJ C00085 BC00085 VJ=100.00  +MOVJ EC00085 VJ=100.00
'Path S3539
SFTOF3D
MOVJ C00086 BC00086 VJ=100.00  +MOVJ EC00086 VJ=100.00
MOVL C00087 BC00087 V=400.0  +MOVJ EC00087 VJ=100.00
SMOVL C00088 BC00088 V=100.0  +MOVJ EC00088
SREFP 3 C00089 BC00089  +REFP EC00089
CALL JOB:SEARCH-R1-S13D
SET P046 P006
SFTON3D P046
SMOVL C00090 BC00090 V=100.0  +MOVJ EC00090
SREFP 3 C00091 BC00091  +REFP EC00091
CALL JOB:SEARCH-R1-S13D
SET P046 P006
SFTON3D P046
SMOVL C00092 BC00092 V=100.0  +MOVJ EC00092
MOVL C00093 BC00093 V=400.0  +MOVJ EC00093 VJ=100.00
MOVL C00094 BC00094 V=1000.0  +MOVJ EC00094 VJ=100.00
'Path S3540
SFTOF3D
MOVJ C00095 BC00095 VJ=100.00  +MOVJ EC00095 VJ=100.00
MOVL C00096 BC00096 V=400.0  +MOVJ EC00096 VJ=100.00
SMOVL C00097 BC00097 V=100.0  +MOVJ EC00097
SREFP 3 C00098 BC00098  +REFP EC00098
CALL JOB:SEARCH-R1-S13D
SET P045 P006
SFTON3D P045
SMOVL C00099 BC00099 V=100.0  +MOVJ EC00099
SREFP 3 C00100 BC00100  +REFP EC00100
CALL JOB:SEARCH-R1-S13D
SET P045 P006
SFTON3D P045
SMOVL C00101 BC00101 V=100.0  +MOVJ EC00101
SREFP 3 C00102 BC00102  +REFP EC00102
CALL JOB:SEARCH-R1-S13D
SET P045 P006
SFTON3D P045
SMOVL C00103 BC00103 V=100.0  +MOVJ EC00103
MOVL C00104 BC00104 V=400.0  +MOVJ EC00104 VJ=100.00
MOVL C00105 BC00105 V=1000.0  +MOVJ EC00105 VJ=100.00
MOVL C00106 BC00106 V=1000.0  +MOVJ EC00106 VJ=100.00
MOVJ C00107 BC00107 VJ=100.00  +MOVJ EC00107 VJ=50.00
SFTOF3D
MOVJ C00108 BC00108 VJ=100.00  +MOVJ EC00108 VJ=50.00
MOVJ C00109 BC00109 VJ=100.00  +MOVJ EC00109 VJ=100.00
MOVL C00110 BC00110 V=400.0  +MOVJ EC00110 VJ=100.00
SMOVL C00111 BC00111 V=100.0  +MOVJ EC00111
SREFP 3 C00112 BC00112  +REFP EC00112
CALL JOB:SEARCH-R1-S13D
SET P043 P006
SFTON3D P043
SMOVL C00113 BC00113 V=100.0  +MOVJ EC00113
SREFP 3 C00114 BC00114  +REFP EC00114
CALL JOB:SEARCH-R1-S13D
SET P043 P006
SFTON3D P043
SMOVL C00115 BC00115 V=100.0  +MOVJ EC00115
SREFP 3 C00116 BC00116  +REFP EC00116
CALL JOB:SEARCH-R1-S13D
SET P043 P006
SFTON3D P043
SMOVL C00117 BC00117 V=100.0  +MOVJ EC00117
MOVL C00118 BC00118 V=400.0  +MOVJ EC00118 VJ=100.00
MOVL C00119 BC00119 V=1000.0  +MOVJ EC00119 VJ=100.00
'Path S3543
SFTOF3D
MOVJ C00120 BC00120 VJ=100.00  +MOVJ EC00120 VJ=100.00
MOVL C00121 BC00121 V=400.0  +MOVJ EC00121 VJ=100.00
SMOVL C00122 BC00122 V=100.0  +MOVJ EC00122
SREFP 3 C00123 BC00123  +REFP EC00123
CALL JOB:SEARCH-R1-S13D
SET P042 P006
SFTON3D P042
SMOVL C00124 BC00124 V=100.0  +MOVJ EC00124
SREFP 3 C00125 BC00125  +REFP EC00125
CALL JOB:SEARCH-R1-S13D
SET P042 P006
SFTON3D P042
SMOVL C00126 BC00126 V=100.0  +MOVJ EC00126
SREFP 3 C00127 BC00127  +REFP EC00127
CALL JOB:SEARCH-R1-S13D
SET P042 P006
SFTON3D P042
SMOVL C00128 BC00128 V=100.0  +MOVJ EC00128
MOVL C00129 BC00129 V=1000.0  +MOVJ EC00129 VJ=100.00
'Path S3544
SFTOF3D
MOVJ C00130 BC00130 VJ=100.00  +MOVJ EC00130 VJ=100.00
MOVL C00131 BC00131 V=400.0  +MOVJ EC00131 VJ=100.00
SMOVL C00132 BC00132 V=100.0  +MOVJ EC00132
SREFP 3 C00133 BC00133  +REFP EC00133
CALL JOB:SEARCH-R1-S13D
SET P041 P006
SFTON3D P041
SMOVL C00134 BC00134 V=100.0  +MOVJ EC00134
SREFP 3 C00135 BC00135  +REFP EC00135
CALL JOB:SEARCH-R1-S13D
SET P041 P006
SFTON3D P041
SMOVL C00136 BC00136 V=100.0  +MOVJ EC00136
SREFP 3 C00137 BC00137  +REFP EC00137
CALL JOB:SEARCH-R1-S13D
SET P041 P006
SFTON3D P041
SMOVL C00138 BC00138 V=100.0  +MOVJ EC00138
MOVL C00139 BC00139 V=400.0  +MOVJ EC00139 VJ=100.00
MOVL C00140 BC00140 V=1000.0  +MOVJ EC00140 VJ=100.00
'Path W3545
SFTOF3D
SFTON3D P041
MOVJ C00141 BC00141 VJ=100.00  +MOVJ EC00141 VJ=100.00
SMOVL C00142 BC00142 V=400.0  +MOVJ EC00142
SMOVL C00143 BC00143 V=133.3 PL=0  +MOVJ EC00143
SREFP 1 C00144 BC00144  +REFP EC00144
SREFP 2 C00145 BC00145  +REFP EC00145
MACRO1 MJ#(0) ARGF9
ARCON
SWVON WEV#(61)
SMOVL C00146 BC00146 V=6.7  +MOVJ EC00146
SMOVL C00147 BC00147 V=6.7  +MOVJ EC00147
SMOVL C00148 BC00148 V=6.7  +MOVJ EC00148
ARCOF
SWVOF
SMOVL C00149 BC00149 V=400.0  +MOVJ EC00149
SMOVL C00150 BC00150 V=1000.0  +MOVJ EC00150
SFTOF3D
'Path W3546
SFTOF3D
SFTON3D P042
MOVJ C00151 BC00151 VJ=100.00  +MOVJ EC00151 VJ=100.00
MOVJ C00152 BC00152 VJ=100.00  +MOVJ EC00152 VJ=100.00
SMOVL C00153 BC00153 V=400.0  +MOVJ EC00153
SMOVL C00154 BC00154 V=133.3 PL=0  +MOVJ EC00154
SREFP 1 C00155 BC00155  +REFP EC00155
SREFP 2 C00156 BC00156  +REFP EC00156
MACRO1 MJ#(0) ARGF14
ARCON
SMOVL C00157 BC00157 V=8.3  +MOVJ EC00157
SMOVL C00158 BC00158 V=8.3  +MOVJ EC00158
SMOVL C00159 BC00159 V=8.3  +MOVJ EC00159
ARCOF
SMOVL C00160 BC00160 V=400.0  +MOVJ EC00160
SMOVL C00161 BC00161 V=333.3  +MOVJ EC00161
SFTOF3D
MOVJ C00162 BC00162 VJ=100.00  +MOVJ EC00162 VJ=100.00
'Path W3547
SFTOF3D
SFTON3D P043
MOVJ C00163 BC00163 VJ=100.00  +MOVJ EC00163 VJ=100.00
MOVJ C00164 BC00164 VJ=100.00  +MOVJ EC00164 VJ=100.00
SMOVL C00165 BC00165 V=400.0  +MOVJ EC00165
SMOVL C00166 BC00166 V=133.3 PL=0  +MOVJ EC00166
SREFP 1 C00167 BC00167  +REFP EC00167
SREFP 2 C00168 BC00168  +REFP EC00168
MACRO1 MJ#(0) ARGF14
ARCON
SMOVL C00169 BC00169 V=8.3  +MOVJ EC00169
SMOVL C00170 BC00170 V=8.3  +MOVJ EC00170
ARCOF
SMOVL C00171 BC00171 V=400.0  +MOVJ EC00171
SMOVL C00172 BC00172 V=1000.0  +MOVJ EC00172
SMOVL C00173 BC00173 V=1000.0  +MOVJ EC00173
SFTOF3D
'NIE SPAWAMY
COMM 'Path W3548
COMM SFTOF3D
COMM SFTON3D P044
COMM MOVJ C00174 BC00174 VJ=100.00  +MOVJ EC00174 VJ=100.00
COMM SMOVL C00175 BC00175 V=400.0  +MOVJ EC00175
COMM SMOVL C00176 BC00176 V=100.0 PL=0  +MOVJ EC00176
COMM SREFP 1 C00177 BC00177  +REFP EC00177
COMM SREFP 2 C00178 BC00178  +REFP EC00178
COMM MACRO1 MJ#(0) ARGF0
COMM ARCON
COMM SMOVL C00179 BC00179 V=10.0  +MOVJ EC00179
COMM SMOVL C00180 BC00180 V=10.0  +MOVJ EC00180
COMM SMOVL C00181 BC00181 V=10.0  +MOVJ EC00181
COMM SMOVL C00182 BC00182 V=10.0  +MOVJ EC00182
COMM SMOVL C00183 BC00183 V=10.0  +MOVJ EC00183
COMM SMOVL C00184 BC00184 V=10.0  +MOVJ EC00184
COMM SMOVL C00185 BC00185 V=10.0  +MOVJ EC00185
COMM SMOVL C00186 BC00186 V=10.0  +MOVJ EC00186
COMM SMOVL C00187 BC00187 V=10.0  +MOVJ EC00187
COMM SMOVL C00188 BC00188 V=10.0  +MOVJ EC00188
COMM SMOVL C00189 BC00189 V=10.0  +MOVJ EC00189
COMM SMOVL C00190 BC00190 V=10.0  +MOVJ EC00190
COMM SMOVL C00191 BC00191 V=10.0  +MOVJ EC00191
COMM SMOVL C00192 BC00192 V=10.0  +MOVJ EC00192
COMM SMOVL C00193 BC00193 V=10.0  +MOVJ EC00193
COMM SMOVL C00194 BC00194 V=10.0  +MOVJ EC00194
COMM SMOVL C00195 BC00195 V=10.0  +MOVJ EC00195
COMM SMOVL C00196 BC00196 V=10.0  +MOVJ EC00196
COMM SMOVL C00197 BC00197 V=10.0  +MOVJ EC00197
COMM SMOVL C00198 BC00198 V=10.0  +MOVJ EC00198
COMM SMOVL C00199 BC00199 V=10.0  +MOVJ EC00199
COMM SMOVL C00200 BC00200 V=10.0  +MOVJ EC00200
COMM SMOVL C00201 BC00201 V=10.0  +MOVJ EC00201
COMM SMOVL C00202 BC00202 V=10.0  +MOVJ EC00202
COMM SMOVL C00203 BC00203 V=10.0  +MOVJ EC00203
COMM ARCOF
COMM SMOVL C00204 BC00204 V=400.0  +MOVJ EC00204
COMM SMOVL C00205 BC00205 V=1000.0  +MOVJ EC00205
COMM SFTOF3D
'Path W3549
SFTOF3D
MOVJ C00206 BC00206 VJ=100.00  +MOVJ EC00206 VJ=100.00
MOVJ C00207 BC00207 VJ=100.00  +MOVJ EC00207 VJ=100.00
SFTON3D P045
MOVJ C00208 BC00208 VJ=100.00  +MOVJ EC00208 VJ=100.00
SMOVL C00209 BC00209 V=400.0  +MOVJ EC00209
SMOVL C00210 BC00210 V=100.0 PL=0  +MOVJ EC00210
SREFP 1 C00211 BC00211  +REFP EC00211
SREFP 2 C00212 BC00212  +REFP EC00212
MACRO1 MJ#(0) ARGF14
ARCON
SMOVL C00213 BC00213 V=8.3  +MOVJ EC00213
SMOVL C00214 BC00214 V=8.3  +MOVJ EC00214
SMOVL C00215 BC00215 V=8.3  +MOVJ EC00215
SMOVL C00216 BC00216 V=8.3  +MOVJ EC00216
SMOVL C00217 BC00217 V=8.3  +MOVJ EC00217
ARCOF
SMOVL C00218 BC00218 V=400.0  +MOVJ EC00218
SMOVL C00219 BC00219 V=1000.0  +MOVJ EC00219
SMOVL C00220 BC00220 V=1000.0  +MOVJ EC00220
MOVJ C00221 BC00221 VJ=100.00  +MOVJ EC00221 VJ=50.00
SFTOF3D
'Path W3550
SFTOF3D
SFTON3D P046
MOVJ C00222 BC00222 VJ=100.00  +MOVJ EC00222 VJ=100.00
MOVJ C00223 BC00223 VJ=100.00  +MOVJ EC00223 VJ=100.00
SMOVL C00224 BC00224 V=400.0  +MOVJ EC00224
SMOVL C00225 BC00225 V=100.0 PL=0  +MOVJ EC00225
SREFP 1 C00226 BC00226  +REFP EC00226
SREFP 2 C00227 BC00227  +REFP EC00227
MACRO1 MJ#(0) ARGF14
ARCON
SMOVL C00228 BC00228 V=8.3  +MOVJ EC00228
SMOVL C00229 BC00229 V=8.3  +MOVJ EC00229
SMOVL C00230 BC00230 V=8.3  +MOVJ EC00230
SMOVL C00231 BC00231 V=8.3  +MOVJ EC00231
SMOVL C00232 BC00232 V=8.3  +MOVJ EC00232
SMOVL C00233 BC00233 V=8.3  +MOVJ EC00233
ARCOF
SMOVL C00234 BC00234 V=400.0  +MOVJ EC00234
SMOVL C00235 BC00235 V=1000.0  +MOVJ EC00235
SFTOF3D
MOVJ C00236 BC00236 VJ=100.00  +MOVJ EC00236 VJ=100.00
MOVJ C00237 BC00237 VJ=100.00  +MOVJ EC00237 VJ=100.00
MOVJ C00238 BC00238 VJ=100.00  +MOVJ EC00238 VJ=100.00
'Down
'Path W3551
SFTOF3D
MOVJ C00239 BC00239 VJ=100.00  +MOVJ EC00239 VJ=100.00
MOVL C00240 BC00240 V=400.0  +MOVJ EC00240 VJ=100.00
SFTON3D P032
SMOVL C00241 BC00241 V=100.0 PL=0  +MOVJ EC00241
SREFP 1 C00242 BC00242  +REFP EC00242
SREFP 2 C00243 BC00243  +REFP EC00243
MACRO1 MJ#(0) ARGF21
ARCON
SWVON WEV#(100)
SMOVC C00244 BC00244 V=9.2  +MOVJ EC00244
SMOVC C00245 BC00245 V=9.2  +MOVJ EC00245
SMOVC C00246 BC00246 V=9.2  +MOVJ EC00246
SMOVC C00247 BC00247 V=9.2  +MOVJ EC00247
SMOVC C00248 BC00248 V=9.2  +MOVJ EC00248
ARCOF
SFTOF3D
SWVOF
MOVL C00249 BC00249 V=400.0  +MOVJ EC00249 VJ=100.00
MOVL C00250 BC00250 V=1000.0  +MOVJ EC00250 VJ=100.00
MOVJ C00251 BC00251 VJ=100.00  +MOVJ EC00251 VJ=100.00
MOVJ C00252 BC00252 VJ=100.00  +MOVJ EC00252 VJ=100.00
MOVJ C00253 BC00253 VJ=100.00  +MOVJ EC00253 VJ=100.00
'Path W3552
SFTOF3D
MOVJ C00254 BC00254 VJ=100.00  +MOVJ EC00254 VJ=100.00
COMM PAUSE
COMM SFTON3D P022
COMM MOVJ C00255 BC00255 VJ=100.00  +MOVJ EC00255 VJ=100.00
COMM SMOVL C00256 BC00256 V=333.3  +MOVJ EC00256
COMM SMOVL C00257 BC00257 V=133.3 PL=0  +MOVJ EC00257
COMM SREFP 1 C00258 BC00258  +REFP EC00258
COMM SREFP 2 C00259 BC00259  +REFP EC00259
COMM MACRO1 MJ#(0) ARGF14
COMM ARCON
COMM SMOVC C00260 BC00260 V=8.3  +MOVJ EC00260
COMM SMOVC C00261 BC00261 V=8.3  +MOVJ EC00261
COMM SMOVC C00262 BC00262 V=8.3  +MOVJ EC00262
COMM SMOVC C00263 BC00263 V=8.3  +MOVJ EC00263
COMM SMOVC C00264 BC00264 V=8.3  +MOVJ EC00264
COMM SMOVC C00265 BC00265 V=8.3  +MOVJ EC00265
COMM SMOVL C00266 BC00266 V=8.3  +MOVJ EC00266
COMM ARCOF
COMM SMOVL C00267 BC00267 V=400.0  +MOVJ EC00267
COMM SMOVL C00268 BC00268 V=1000.0  +MOVJ EC00268
COMM SFTOF3D
COMM 'Path W3553
COMM SFTOF3D
COMM SFTON3D P022
COMM MOVJ C00269 BC00269 VJ=100.00  +MOVJ EC00269 VJ=100.00
COMM SMOVL C00270 BC00270 V=133.3  +MOVJ EC00270
COMM 'SZEROKA SZCZELINA!!!
COMM MACRO1 MJ#(0) ARGF14
COMM SMOVL C00271 BC00271 V=133.3 PL=0  +MOVJ EC00271
COMM SREFP 1 C00272 BC00272  +REFP EC00272
COMM SREFP 2 C00273 BC00273  +REFP EC00273
COMM ARCON
COMM SWVON WEV#(14)
COMM SMOVL C00274 BC00274 V=7.5  +MOVJ EC00274
COMM SMOVL C00275 BC00275 V=7.5  +MOVJ EC00275
COMM ARCOF
COMM SWVOF
COMM SMOVL C00276 BC00276 V=400.0  +MOVJ EC00276
COMM SFTOF3D
COMM PAUSE
SMOVL C00277 BC00277 V=1000.0  +MOVJ EC00277
MOVJ C00278 BC00278 VJ=70.00  +MOVJ EC00278 VJ=70.00
MACRO1 MJ#(0) ARGF14
SFTON3D P088
SMOVL C00279 BC00279 V=166.7  +MOVJ EC00279
ARCON
SMOVL C00280 BC00280 V=10.8  +MOVJ EC00280
ARCOF
SFTOF3D
SMOVL C00281 BC00281 V=250.0  +MOVJ EC00281
'
'NIE SPAWAMY_BRAK BLASZKI
COMM 'Path W3554
COMM SFTOF3D
COMM SFTON3D P023
COMM MOVJ C00282 BC00282 VJ=100.00  +MOVJ EC00282 VJ=100.00
COMM MOVJ C00283 BC00283 VJ=100.00  +MOVJ EC00283 VJ=100.00
COMM SMOVL C00284 BC00284 V=400.0  +MOVJ EC00284
COMM SMOVL C00285 BC00285 V=100.0 PL=0  +MOVJ EC00285
COMM SREFP 1 C00286 BC00286  +REFP EC00286
COMM SREFP 2 C00287 BC00287  +REFP EC00287
COMM MACRO1 MJ#(0) ARGF0
COMM ARCON
COMM SMOVL C00288 BC00288 V=10.0  +MOVJ EC00288
COMM SMOVL C00289 BC00289 V=10.0  +MOVJ EC00289
COMM SMOVL C00290 BC00290 V=10.0  +MOVJ EC00290
COMM ARCOF
COMM SMOVL C00291 BC00291 V=400.0  +MOVJ EC00291
COMM SMOVL C00292 BC00292 V=1000.0  +MOVJ EC00292
COMM SFTOF3D
COMM MOVJ C00293 BC00293 VJ=100.00  +MOVJ EC00293 VJ=100.00
'NIE SPAWAMY_BRAK BLASZKI
COMM 'Path W3555
COMM SFTOF3D
COMM SFTON3D P023
COMM MOVJ C00294 BC00294 VJ=100.00  +MOVJ EC00294 VJ=100.00
COMM SMOVL C00295 BC00295 V=100.0  +MOVJ EC00295
COMM SMOVL C00296 BC00296 V=100.0 PL=0  +MOVJ EC00296
COMM SREFP 1 C00297 BC00297  +REFP EC00297
COMM SREFP 2 C00298 BC00298  +REFP EC00298
COMM MACRO1 MJ#(0) ARGF0
COMM ARCON
COMM SMOVL C00299 BC00299 V=10.0  +MOVJ EC00299
COMM SMOVL C00300 BC00300 V=10.0  +MOVJ EC00300
COMM SMOVL C00301 BC00301 V=10.0  +MOVJ EC00301
COMM ARCOF
COMM SMOVL C00302 BC00302 V=400.0  +MOVJ EC00302
COMM SMOVL C00303 BC00303 V=1000.0  +MOVJ EC00303
COMM SMOVL C00304 BC00304 V=1000.0  +MOVJ EC00304
COMM SFTOF3D
'NIE SPAWAMY_BRAK BLASZKI
COMM 'Path W3556
COMM SFTOF3D
COMM SFTON3D P023
COMM MOVJ C00305 BC00305 VJ=100.00  +MOVJ EC00305 VJ=100.00
COMM SMOVL C00306 BC00306 V=100.0  +MOVJ EC00306
COMM SMOVL C00307 BC00307 V=100.0 PL=0  +MOVJ EC00307
COMM SREFP 1 C00308 BC00308  +REFP EC00308
COMM SREFP 2 C00309 BC00309  +REFP EC00309
COMM MACRO1 MJ#(0) ARGF0
COMM ARCON
COMM SMOVL C00310 BC00310 V=10.0  +MOVJ EC00310
COMM ARCOF
COMM SMOVL C00311 BC00311 V=400.0  +MOVJ EC00311
COMM SMOVL C00312 BC00312 V=1000.0  +MOVJ EC00312
COMM SFTOF3D
'
'NIE SPAWAMY_BRAK BLASZKI
COMM 'Path W3557
COMM SFTOF3D
COMM SFTON3D P024
COMM MOVJ C00313 BC00313 VJ=100.00  +MOVJ EC00313 VJ=100.00
COMM SMOVL C00314 BC00314 V=100.0  +MOVJ EC00314
COMM SMOVL C00315 BC00315 V=100.0 PL=0  +MOVJ EC00315
COMM SREFP 1 C00316 BC00316  +REFP EC00316
COMM SREFP 2 C00317 BC00317  +REFP EC00317
COMM MACRO1 MJ#(0) ARGF0
COMM ARCON
COMM SMOVL C00318 BC00318 V=10.0  +MOVJ EC00318
COMM SMOVL C00319 BC00319 V=10.0  +MOVJ EC00319
COMM SMOVL C00320 BC00320 V=10.0  +MOVJ EC00320
COMM ARCOF
COMM SMOVL C00321 BC00321 V=400.0  +MOVJ EC00321
COMM SMOVL C00322 BC00322 V=1000.0  +MOVJ EC00322
COMM SFTOF3D
COMM MOVJ C00323 BC00323 VJ=100.00  +MOVJ EC00323 VJ=100.00
'NIE SPAWAMY_BRAK BLASZKI
COMM 'Path W3558
COMM SFTOF3D
COMM SFTON3D P024
COMM MOVJ C00324 BC00324 VJ=100.00  +MOVJ EC00324 VJ=100.00
COMM SMOVL C00325 BC00325 V=100.0  +MOVJ EC00325
COMM SMOVL C00326 BC00326 V=100.0 PL=0  +MOVJ EC00326
COMM SREFP 1 C00327 BC00327  +REFP EC00327
COMM SREFP 2 C00328 BC00328  +REFP EC00328
COMM MACRO1 MJ#(0) ARGF0
COMM ARCON
COMM SMOVL C00329 BC00329 V=10.0  +MOVJ EC00329
COMM SMOVL C00330 BC00330 V=10.0  +MOVJ EC00330
COMM SMOVL C00331 BC00331 V=10.0  +MOVJ EC00331
COMM ARCOF
COMM SMOVL C00332 BC00332 V=400.0  +MOVJ EC00332
COMM SMOVL C00333 BC00333 V=1000.0  +MOVJ EC00333
COMM SMOVL C00334 BC00334 V=1000.0  +MOVJ EC00334
COMM SFTOF3D
'NIE SPAWAMY_BRAK BLASZKI
COMM 'Path W3559
COMM SFTOF3D
COMM SFTON3D P024
COMM MOVJ C00335 BC00335 VJ=100.00  +MOVJ EC00335 VJ=100.00
COMM SMOVL C00336 BC00336 V=100.0  +MOVJ EC00336
COMM SMOVL C00337 BC00337 V=100.0 PL=0  +MOVJ EC00337
COMM SREFP 1 C00338 BC00338  +REFP EC00338
COMM SREFP 2 C00339 BC00339  +REFP EC00339
COMM MACRO1 MJ#(0) ARGF0
COMM ARCON
COMM SMOVL C00340 BC00340 V=10.0  +MOVJ EC00340
COMM ARCOF
COMM SMOVL C00341 BC00341 V=400.0  +MOVJ EC00341
COMM SMOVL C00342 BC00342 V=1000.0  +MOVJ EC00342
COMM SFTOF3D
COMM MOVJ C00343 BC00343 VJ=100.00  +MOVJ EC00343 VJ=100.00
'
'NIE SPAWAMY_BRAK BLASZKI
COMM 'Path W3560
COMM SFTOF3D
COMM SFTON3D P025
COMM MOVJ C00344 BC00344 VJ=100.00  +MOVJ EC00344 VJ=100.00
COMM SMOVL C00345 BC00345 V=100.0  +MOVJ EC00345
COMM SMOVL C00346 BC00346 V=100.0 PL=0  +MOVJ EC00346
COMM SREFP 1 C00347 BC00347  +REFP EC00347
COMM SREFP 2 C00348 BC00348  +REFP EC00348
COMM MACRO1 MJ#(0) ARGF0
COMM ARCON
COMM SMOVL C00349 BC00349 V=10.0  +MOVJ EC00349
COMM SMOVL C00350 BC00350 V=10.0  +MOVJ EC00350
COMM SMOVL C00351 BC00351 V=10.0  +MOVJ EC00351
COMM ARCOF
COMM SMOVL C00352 BC00352 V=400.0  +MOVJ EC00352
COMM SMOVL C00353 BC00353 V=1000.0  +MOVJ EC00353
COMM SFTOF3D
COMM MOVJ C00354 BC00354 VJ=100.00  +MOVJ EC00354 VJ=100.00
'NIE SPAWAMY_BRAK BLASZKI
COMM 'Path W3561
COMM SFTOF3D
COMM SFTON3D P025
COMM MOVJ C00355 BC00355 VJ=100.00  +MOVJ EC00355 VJ=100.00
COMM SMOVL C00356 BC00356 V=100.0  +MOVJ EC00356
COMM SMOVL C00357 BC00357 V=100.0 PL=0  +MOVJ EC00357
COMM SREFP 1 C00358 BC00358  +REFP EC00358
COMM SREFP 2 C00359 BC00359  +REFP EC00359
COMM MACRO1 MJ#(0) ARGF0
COMM ARCON
COMM SMOVL C00360 BC00360 V=10.0  +MOVJ EC00360
COMM SMOVL C00361 BC00361 V=10.0  +MOVJ EC00361
COMM SMOVL C00362 BC00362 V=10.0  +MOVJ EC00362
COMM ARCOF
COMM SMOVL C00363 BC00363 V=400.0  +MOVJ EC00363
COMM SMOVL C00364 BC00364 V=1000.0  +MOVJ EC00364
COMM SMOVL C00365 BC00365 V=1000.0  +MOVJ EC00365
COMM SFTOF3D
'NIE SPAWAMY_BRAK BLASZKI
COMM 'Path W3562
COMM SFTOF3D
COMM SFTON3D P025
COMM MOVJ C00366 BC00366 VJ=100.00  +MOVJ EC00366 VJ=100.00
COMM SMOVL C00367 BC00367 V=100.0  +MOVJ EC00367
COMM SMOVL C00368 BC00368 V=100.0 PL=0  +MOVJ EC00368
COMM SREFP 1 C00369 BC00369  +REFP EC00369
COMM SREFP 2 C00370 BC00370  +REFP EC00370
COMM MACRO1 MJ#(0) ARGF0
COMM ARCON
COMM SMOVL C00371 BC00371 V=10.0  +MOVJ EC00371
COMM ARCOF
COMM SMOVL C00372 BC00372 V=400.0  +MOVJ EC00372
COMM SMOVL C00373 BC00373 V=1000.0  +MOVJ EC00373
COMM SFTOF3D
COMM MOVJ C00374 BC00374 VJ=100.00  +MOVJ EC00374 VJ=100.00
COMM MOVJ C00375 BC00375 VJ=100.00  +MOVJ EC00375 VJ=100.00
COMM '
COMM MOVJ C00376 BC00376 VJ=100.00  +MOVJ EC00376 VJ=100.00
COMM MOVJ C00377 BC00377 VJ=100.00  +MOVJ EC00377 VJ=100.00
'NIE SPAWAMY_BRAK BLASZKI
COMM 'Path W3563
COMM SFTOF3D
COMM SFTON3D P023
COMM MOVJ C00378 BC00378 VJ=100.00  +MOVJ EC00378 VJ=100.00
COMM SMOVL C00379 BC00379 V=400.0  +MOVJ EC00379
COMM SMOVL C00380 BC00380 V=100.0 PL=0  +MOVJ EC00380
COMM SREFP 1 C00381 BC00381  +REFP EC00381
COMM SREFP 2 C00382 BC00382  +REFP EC00382
COMM MACRO1 MJ#(0) ARGF0
COMM ARCON
COMM SMOVL C00383 BC00383 V=10.0  +MOVJ EC00383
COMM SMOVL C00384 BC00384 V=10.0  +MOVJ EC00384
COMM SMOVL C00385 BC00385 V=10.0  +MOVJ EC00385
COMM ARCOF
COMM SMOVL C00386 BC00386 V=400.0  +MOVJ EC00386
COMM SMOVL C00387 BC00387 V=1000.0  +MOVJ EC00387
COMM SMOVL C00388 BC00388 V=1000.0  +MOVJ EC00388
COMM SFTOF3D
'NIE SPAWAMY_BRAK BLASZKI
COMM 'Path W3564
COMM SFTOF3D
COMM SFTON3D P023
COMM SMOVL C00389 BC00389 V=100.0  +MOVJ EC00389
COMM SMOVL C00390 BC00390 V=100.0 PL=0  +MOVJ EC00390
COMM SREFP 1 C00391 BC00391  +REFP EC00391
COMM SREFP 2 C00392 BC00392  +REFP EC00392
COMM MACRO1 MJ#(0) ARGF0
COMM ARCON
COMM SMOVL C00393 BC00393 V=10.0  +MOVJ EC00393
COMM SMOVL C00394 BC00394 V=10.0  +MOVJ EC00394
COMM SMOVL C00395 BC00395 V=10.0  +MOVJ EC00395
COMM ARCOF
COMM SMOVL C00396 BC00396 V=400.0  +MOVJ EC00396
COMM SFTOF3D
COMM MOVJ C00397 BC00397 VJ=100.00  +MOVJ EC00397 VJ=100.00
'
COMM MOVJ C00398 BC00398 VJ=100.00  +MOVJ EC00398 VJ=100.00
'NIE SPAWAMY_BRAK BLASZKI
COMM 'Path W3565
COMM SFTOF3D
COMM SFTON3D P024
COMM MOVJ C00399 BC00399 VJ=100.00  +MOVJ EC00399 VJ=100.00
COMM MOVJ C00400 BC00400 VJ=100.00  +MOVJ EC00400 VJ=100.00
COMM SMOVL C00401 BC00401 V=400.0  +MOVJ EC00401
COMM SMOVL C00402 BC00402 V=100.0 PL=0  +MOVJ EC00402
COMM SREFP 1 C00403 BC00403  +REFP EC00403
COMM SREFP 2 C00404 BC00404  +REFP EC00404
COMM MACRO1 MJ#(0) ARGF0
COMM ARCON
COMM SMOVL C00405 BC00405 V=10.0  +MOVJ EC00405
COMM SMOVL C00406 BC00406 V=10.0  +MOVJ EC00406
COMM SMOVL C00407 BC00407 V=10.0  +MOVJ EC00407
COMM ARCOF
COMM SMOVL C00408 BC00408 V=400.0  +MOVJ EC00408
COMM SMOVL C00409 BC00409 V=1000.0  +MOVJ EC00409
COMM SMOVL C00410 BC00410 V=1000.0  +MOVJ EC00410
COMM SFTOF3D
'NIE SPAWAMY_BRAK BLASZKI
COMM 'Path W3566
COMM SFTOF3D
COMM SFTON3D P025
COMM MOVJ C00411 BC00411 VJ=100.00  +MOVJ EC00411 VJ=100.00
COMM SMOVL C00412 BC00412 V=400.0  +MOVJ EC00412
COMM SMOVL C00413 BC00413 V=100.0 PL=0  +MOVJ EC00413
COMM SREFP 1 C00414 BC00414  +REFP EC00414
COMM SREFP 2 C00415 BC00415  +REFP EC00415
COMM MACRO1 MJ#(0) ARGF0
COMM ARCON
COMM SMOVL C00416 BC00416 V=10.0  +MOVJ EC00416
COMM SMOVL C00417 BC00417 V=10.0  +MOVJ EC00417
COMM SMOVL C00418 BC00418 V=10.0  +MOVJ EC00418
COMM ARCOF
COMM SMOVL C00419 BC00419 V=400.0  +MOVJ EC00419
COMM SMOVL C00420 BC00420 V=1000.0  +MOVJ EC00420
COMM SMOVL C00421 BC00421 V=1000.0  +MOVJ EC00421
COMM SFTOF3D
MOVJ C00422 BC00422 VJ=100.00  +MOVJ EC00422 VJ=100.00
MOVJ C00423 BC00423 VJ=100.00  +MOVJ EC00423 VJ=50.00
MOVJ C00424 BC00424 VJ=100.00  +MOVJ EC00424 VJ=50.00
MOVJ C00425 BC00425 VJ=100.00  +MOVJ EC00425 VJ=50.00
MOVJ C00426 BC00426 VJ=100.00  +MOVJ EC00426 VJ=100.00
'Path W3567
SFTOF3D
SFTON3D P021
MOVJ C00427 BC00427 VJ=100.00  +MOVJ EC00427 VJ=100.00
SMOVL C00428 BC00428 V=250.0  +MOVJ EC00428
SMOVL C00429 BC00429 V=133.3 PL=0  +MOVJ EC00429
SREFP 1 C00430 BC00430  +REFP EC00430
SREFP 2 C00431 BC00431  +REFP EC00431
MACRO1 MJ#(0) ARGF21
ARCON
SWVON WEV#(100)
SMOVC C00432 BC00432 V=9.2  +MOVJ EC00432
SMOVC C00433 BC00433 V=9.2  +MOVJ EC00433
SMOVC C00434 BC00434 V=9.2  +MOVJ EC00434
SMOVC C00435 BC00435 V=9.2  +MOVJ EC00435
ARCOF
SWVOF
SMOVL C00436 BC00436 V=400.0  +MOVJ EC00436
SMOVL C00437 BC00437 V=1000.0  +MOVJ EC00437
SFTOF3D
MOVJ C00438 BC00438 VJ=100.00  +MOVJ EC00438 VJ=100.00
'
MOVJ C00439 BC00439 VJ=100.00  +MOVJ EC00439 VJ=100.00
MOVJ C00440 BC00440 VJ=100.00  +MOVJ EC00440 VJ=100.00
'NIE SPAWAMY_BRAK BLASZKI
COMM 'Path W3568
COMM SFTOF3D
COMM SFTON3D P024
COMM MOVJ C00441 BC00441 VJ=100.00  +MOVJ EC00441 VJ=100.00
COMM SMOVL C00442 BC00442 V=100.0  +MOVJ EC00442
COMM SMOVL C00443 BC00443 V=100.0 PL=0  +MOVJ EC00443
COMM SREFP 1 C00444 BC00444  +REFP EC00444
COMM SREFP 2 C00445 BC00445  +REFP EC00445
COMM MACRO1 MJ#(0) ARGF0
COMM ARCON
COMM SMOVL C00446 BC00446 V=10.0  +MOVJ EC00446
COMM SMOVL C00447 BC00447 V=10.0  +MOVJ EC00447
COMM SMOVL C00448 BC00448 V=10.0  +MOVJ EC00448
COMM ARCOF
COMM SMOVL C00449 BC00449 V=400.0  +MOVJ EC00449
COMM SMOVL C00450 BC00450 V=1000.0  +MOVJ EC00450
COMM SFTOF3D
'NIE SPAWAMY_BRAK BLASZKI
COMM 'Path W3569
COMM SFTOF3D
COMM SFTON3D P025
COMM MOVJ C00451 BC00451 VJ=100.00  +MOVJ EC00451 VJ=100.00
COMM SMOVL C00452 BC00452 V=100.0  +MOVJ EC00452
COMM SMOVL C00453 BC00453 V=100.0 PL=0  +MOVJ EC00453
COMM SREFP 1 C00454 BC00454  +REFP EC00454
COMM SREFP 2 C00455 BC00455  +REFP EC00455
COMM MACRO1 MJ#(0) ARGF0
COMM ARCON
COMM SMOVL C00456 BC00456 V=10.0  +MOVJ EC00456
COMM SMOVL C00457 BC00457 V=10.0  +MOVJ EC00457
COMM SMOVL C00458 BC00458 V=10.0  +MOVJ EC00458
COMM ARCOF
COMM SMOVL C00459 BC00459 V=400.0  +MOVJ EC00459
COMM SMOVL C00460 BC00460 V=1000.0  +MOVJ EC00460
COMM SMOVL C00461 BC00461 V=1000.0  +MOVJ EC00461
COMM SFTOF3D
COMM MOVJ C00462 BC00462 VJ=100.00  +MOVJ EC00462 VJ=100.00
COMM '
COMM MOVJ C00463 BC00463 VJ=100.00  +MOVJ EC00463 VJ=100.00
COMM MOVJ C00464 BC00464 VJ=100.00  +MOVJ EC00464 VJ=100.00
'Path W3570
SFTOF3D
SFTON3D P026
MOVJ C00465 BC00465 VJ=100.00  +MOVJ EC00465 VJ=100.00
MOVJ C00466 BC00466 VJ=100.00  +MOVJ EC00466 VJ=100.00
SMOVL C00467 BC00467 V=666.7  +MOVJ EC00467
SMOVL C00468 BC00468 V=133.3  +MOVJ EC00468
SREFP 1 C00469 BC00469  +REFP EC00469
SREFP 2 C00470 BC00470  +REFP EC00470
MACRO1 MJ#(0) ARGF21
ARCON
SMOVL C00471 BC00471 V=7.5  +MOVJ EC00471
SMOVL C00472 BC00472 V=7.5  +MOVJ EC00472
SMOVL C00473 BC00473 V=7.5  +MOVJ EC00473
SMOVL C00474 BC00474 V=7.5  +MOVJ EC00474
SMOVL C00475 BC00475 V=7.5  +MOVJ EC00475
SMOVL C00476 BC00476 V=7.5  +MOVJ EC00476
SMOVL C00477 BC00477 V=7.5  +MOVJ EC00477
ARCON
SMOVL C00478 BC00478 V=7.5  +MOVJ EC00478
SMOVL C00479 BC00479 V=7.5  +MOVJ EC00479
SMOVL C00480 BC00480 V=7.5  +MOVJ EC00480
SMOVL C00481 BC00481 V=7.5  +MOVJ EC00481
ARCOF
SMOVL C00482 BC00482 V=250.0  +MOVJ EC00482
SMOVL C00483 BC00483 V=1000.0  +MOVJ EC00483
SFTOF3D
MOVJ C00484 BC00484 VJ=100.00  +MOVJ EC00484 VJ=100.00
'jakie searche do takicj spoin?
MOVJ C00485 BC00485 VJ=100.00  +MOVJ EC00485 VJ=100.00
MOVJ C00486 BC00486 VJ=100.00  +MOVJ EC00486 VJ=100.00
'Path W3572
SFTOF3D
'jakie searche do takicj spoin?
MOVJ C00487 BC00487 VJ=100.00  +MOVJ EC00487 VJ=100.00
'Path W3579
SFTOF3D
MOVJ C00488 BC00488 VJ=50.00  +MOVJ EC00488 VJ=100.00
COMM PAUSE
COMM MOVL C00489 BC00489 V=400.0  +MOVJ EC00489 VJ=100.00
COMM SFTOF3D
COMM SFTON3D P089
COMM SMOVL C00490 BC00490 V=100.0 PL=0  +MOVJ EC00490
COMM SREFP 1 C00491 BC00491  +REFP EC00491
COMM SREFP 2 C00492 BC00492  +REFP EC00492
COMM MACRO1 MJ#(0) ARGF9
COMM ARCON
COMM SMOVL C00493 BC00493 V=11.7  +MOVJ EC00493
COMM ARCOF
COMM MOVL C00494 BC00494 V=666.7  +MOVJ EC00494 VJ=100.00
COMM SMOVL C00495 BC00495 V=166.7  +MOVJ EC00495
COMM ARCON
COMM SMOVL C00496 BC00496 V=11.7  +MOVJ EC00496
COMM ARCOF
COMM SFTOF3D
SMOVL C00497 BC00497 V=250.0  +MOVJ EC00497
MACRO1 MJ#(0) ARGF14
MOVL C00498 BC00498 V=1000.0  +MOVJ EC00498 VJ=100.00
SFTON3D P090
SMOVL C00499 BC00499 V=166.7  +MOVJ EC00499
ARCON
SMOVL C00500 BC00500 V=12.5  +MOVJ EC00500
ARCOF
SMOVL C00501 BC00501 V=166.7  +MOVJ EC00501
SMOVL C00502 BC00502 V=166.7  +MOVJ EC00502
SMOVL C00503 BC00503 V=166.7  +MOVJ EC00503
ARCON
SMOVL C00504 BC00504 V=10.8  +MOVJ EC00504
ARCOF
SMOVL C00505 BC00505 V=166.7  +MOVJ EC00505
SFTOF3D
SMOVL C00506 BC00506 V=1000.0  +MOVJ EC00506
MOVJ C00507 BC00507 VJ=100.00  +MOVJ EC00507 VJ=100.00
COMM MOVJ C00508 BC00508 VJ=100.00  +MOVJ EC00508 VJ=100.00
COMM MOVJ C00509 BC00509 VJ=100.00  +MOVJ EC00509 VJ=100.00
'NIE SPAWAMY
COMM 'Path W3582
COMM SFTOF3D
COMM PAUSE
COMM SFTON3D P031
COMM MOVJ C00510 BC00510 VJ=100.00  +MOVJ EC00510 VJ=100.00
COMM SMOVL C00511 BC00511 V=100.0  +MOVJ EC00511
COMM SMOVL C00512 BC00512 V=100.0 PL=0  +MOVJ EC00512
COMM SREFP 1 C00513 BC00513  +REFP EC00513
COMM SREFP 2 C00514 BC00514  +REFP EC00514
COMM MACRO1 MJ#(0) ARGF0
COMM ARCON
COMM SMOVL C00515 BC00515 V=10.0  +MOVJ EC00515
COMM SMOVL C00516 BC00516 V=10.0  +MOVJ EC00516
COMM SMOVL C00517 BC00517 V=10.0  +MOVJ EC00517
COMM ARCOF
COMM SMOVL C00518 BC00518 V=400.0  +MOVJ EC00518
COMM SMOVL C00519 BC00519 V=1000.0  +MOVJ EC00519
COMM SFTOF3D
'Down
MOVJ C00520 BC00520 VJ=100.00  +MOVJ EC00520 VJ=100.00
END
